	UF : 0, UT : 6,		CONFIG : 'N U T, 0, 0, 0',
	X =  474.797  mm,	Y =   -334.589  mm,	Z =   -248.128  mm,
	W =  90.000 deg,	P =   0.000 deg,	R =   90.000 deg
};
P[1529]{
   GP1:
	UF : 0, UT : 6,		CONFIG : 'N U T, 0, 0, 0',
	X =  474.358  mm,	Y =   -333.597  mm,	Z =   -247.804  mm,
	W =  90.000 deg,	P =   0.000 deg,	R =   90.000 deg
};
P[1530]{
   GP1:
	UF : 0, UT : 6,		CONFIG : 'N U T, 0, 0, 0',
	X =  473.486  mm,	Y =   -332.265  mm,	Z =   -248.052  mm,
	W =  90.000 deg,	P =   0.000 deg,	R =   90.000 deg
};
P[1531]{
   GP1:
	UF : 0, UT : 6,		CONFIG : 'N U T, 0, 0, 0',
	X =  472.911  mm,	Y =   -331.359  mm,	Z =   -248.179  mm,
	W =  90.000 deg,	P =   0.000 deg,	R =   90.000 deg
};
P[1532]{
   GP1:
	UF : 0, UT : 6,		CONFIG : 'N U T, 0, 0, 0',
	X =  472.436  mm,	Y =   -330.414  mm,	Z =   -248.006  mm,
	W =  90.000 deg,	P =   0.000 deg,	R =   90.000 deg
};
P[1533]{
   GP1:
	UF : 0, UT : 6,		CONFIG : 'N U T, 0, 0, 0',
	X =  470.822  mm,	Y =   -327.714  mm,	Z =   -248.142  mm,
	W =  90.000 deg,	P =   0.000 deg,	R =   90.000 deg
};
P[1534]{
   GP1:
	UF : 0, UT : 6,		CONFIG : 'N U T, 0, 0, 0',
	X =  470.360  mm,	Y =   -326.792  mm,	Z =   -247.970  mm,
	W =  90.000 deg,	P =   0.000 deg,	R =   90.000 deg
};
P[1535]{
   GP1:
	UF : 0, UT : 6,		CONFIG : 'N U T, 0, 0, 0',
	X =  469.532  mm,	Y =   -325.400  mm,	Z =   -248.029  mm,
	W =  90.000 deg,	P =   0.000 deg,	R =   90.000 deg
};
P[1536]{
   GP1:
	UF : 0, UT : 6,		CONFIG : 'N U T, 0, 0, 0',
	X =  468.396  mm,	Y =   -323.373  mm,	Z =   -247.945  mm,
	W =  90.000 deg,	P =   0.000 deg,	R =   90.000 deg
};
P[1537]{
   GP1:
	UF : 0, UT : 6,		CONFIG : 'N U T, 0, 0, 0',
	X =  467.953  mm,	Y =   -322.646  mm,	Z =   -248.001  mm,
	W =  90.000 deg,	P =   0.000 deg,	R =   90.000 deg
};
P[1538]{
   GP1:
	UF : 0, UT : 6,		CONFIG : 'N U T, 0, 0, 0',
	X =  467.093  mm,	Y =   -321.165  mm,	Z =   -248.010  mm,
	W =  90.000 deg,	P =   0.000 deg,	R =   90.000 deg
};
P[1539]{
   GP1:
	UF : 0, UT : 6,		CONFIG : 'N U T, 0, 0, 0',
	X =  465.613  mm,	Y =   -318.699  mm,	Z =   -248.148  mm,
	W =  90.000 deg,	P =   0.000 deg,	R =   90.000 deg
};
P[1540]{
   GP1:
	UF : 0, UT : 6,		CONFIG : 'N U T, 0, 0, 0',
	X =  464.567  mm,	Y =   -316.920  mm,	Z =   -248.196  mm,
	W =  90.000 deg,	P =   0.000 deg,	R =   90.000 deg
};
P[1541]{
   GP1:
	UF : 0, UT : 6,		CONFIG : 'N U T, 0, 0, 0',
	X =  463.631  mm,	Y =   -315.161  mm,	Z =   -248.002  mm,
	W =  90.000 deg,	P =   0.000 deg,	R =   90.000 deg
};
P[1542]{
   GP1:
	UF : 0, UT : 6,		CONFIG : 'N U T, 0, 0, 0',
	X =  463.100  mm,	Y =   -314.216  mm,	Z =   -247.965  mm,
	W =  90.000 deg,	P =   0.000 deg,	R =   90.000 deg
};
P[1543]{
   GP1:
	UF : 0, UT : 6,		CONFIG : 'N U T, 0, 0, 0',
	X =  462.160  mm,	Y =   -312.535  mm,	Z =   -247.892  mm,
	W =  90.000 deg,	P =   0.000 deg,	R =   90.000 deg
};
P[1544]{
   GP1:
	UF : 0, UT : 6,		CONFIG : 'N U T, 0, 0, 0',
	X =  461.282  mm,	Y =   -311.005  mm,	Z =   -247.880  mm,
	W =  90.000 deg,	P =   0.000 deg,	R =   90.000 deg
};
P[1545]{
   GP1:
	UF : 0, UT : 6,		CONFIG : 'N U T, 0, 0, 0',
	X =  460.643  mm,	Y =   -310.130  mm,	Z =   -248.205  mm,
	W =  90.000 deg,	P =   0.000 deg,	R =   90.000 deg
};
P[1546]{
   GP1:
	UF : 0, UT : 6,		CONFIG : 'N U T, 0, 0, 0',
	X =  458.837  mm,	Y =   -307.025  mm,	Z =   -248.237  mm,
	W =  90.000 deg,	P =   0.000 deg,	R =   90.000 deg
};
P[1547]{
   GP1:
	UF : 0, UT : 6,		CONFIG : 'N U T, 0, 0, 0',
	X =  457.547  mm,	Y =   -304.731  mm,	Z =   -248.150  mm,
	W =  90.000 deg,	P =   0.000 deg,	R =   90.000 deg
};
P[1548]{
   GP1:
	UF : 0, UT : 6,		CONFIG : 'N U T, 0, 0, 0',
	X =  456.867  mm,	Y =   -303.518  mm,	Z =   -248.103  mm,
	W =  90.000 deg,	P =   0.000 deg,	R =   90.000 deg
};
P[1549]{
   GP1:
	UF : 0, UT : 6,		CONFIG : 'N U T, 0, 0, 0',
	X =  455.788  mm,	Y =   -301.711  mm,	Z =   -248.187  mm,
	W =  90.000 deg,	P =   0.000 deg,	R =   90.000 deg
};
P[1550]{
   GP1:
	UF : 0, UT : 6,		CONFIG : 'N U T, 0, 0, 0',
	X =  454.454  mm,	Y =   -299.407  mm,	Z =   -248.197  mm,
	W =  90.000 deg,	P =   0.000 deg,	R =   90.000 deg
};
P[1551]{
   GP1:
	UF : 0, UT : 6,		CONFIG : 'N U T, 0, 0, 0',
	X =  453.882  mm,	Y =   -298.356  mm,	Z =   -248.113  mm,
	W =  90.000 deg,	P =   0.000 deg,	R =   90.000 deg
};
P[1552]{
   GP1:
	UF : 0, UT : 6,		CONFIG : 'N U T, 0, 0, 0',
	X =  453.477  mm,	Y =   -297.544  mm,	Z =   -247.960  mm,
	W =  90.000 deg,	P =   0.000 deg,	R =   90.000 deg
};
P[1553]{
   GP1:
	UF : 0, UT : 6,		CONFIG : 'N U T, 0, 0, 0',
	X =  452.176  mm,	Y =   -295.442  mm,	Z =   -248.171  mm,
	W =  90.000 deg,	P =   0.000 deg,	R =   90.000 deg
};
P[1554]{
   GP1:
	UF : 0, UT : 6,		CONFIG : 'N U T, 0, 0, 0',
	X =  451.411  mm,	Y =   -294.155  mm,	Z =   -248.222  mm,
	W =  90.000 deg,	P =   0.000 deg,	R =   90.000 deg
};
P[1555]{
   GP1:
	UF : 0, UT : 6,		CONFIG : 'N U T, 0, 0, 0',
	X =  450.241  mm,	Y =   -291.952  mm,	Z =   -247.976  mm,
	W =  90.000 deg,	P =   0.000 deg,	R =   90.000 deg
};
P[1556]{
   GP1:
	UF : 0, UT : 6,		CONFIG : 'N U T, 0, 0, 0',
	X =  449.232  mm,	Y =   -290.232  mm,	Z =   -248.015  mm,
	W =  90.000 deg,	P =   0.000 deg,	R =   90.000 deg
};
P[1557]{
   GP1:
	UF : 0, UT : 6,		CONFIG : 'N U T, 0, 0, 0',
	X =  448.784  mm,	Y =   -289.434  mm,	Z =   -247.984  mm,
	W =  90.000 deg,	P =   0.000 deg,	R =   90.000 deg
};
P[1558]{
   GP1:
	UF : 0, UT : 6,		CONFIG : 'N U T, 0, 0, 0',
	X =  447.902  mm,	Y =   -288.033  mm,	Z =   -248.160  mm,
	W =  90.000 deg,	P =   0.000 deg,	R =   90.000 deg
};
P[1559]{
   GP1:
	UF : 0, UT : 6,		CONFIG : 'N U T, 0, 0, 0',
	X =  447.571  mm,	Y =   -287.324  mm,	Z =   -247.969  mm,
	W =  90.000 deg,	P =   0.000 deg,	R =   90.000 deg
};
P[1560]{
   GP1:
	UF : 0, UT : 6,		CONFIG : 'N U T, 0, 0, 0',
	X =  445.908  mm,	Y =   -284.546  mm,	Z =   -248.113  mm,
	W =  90.000 deg,	P =   0.000 deg,	R =   90.000 deg
};
P[1561]{
   GP1:
	UF : 0, UT : 6,		CONFIG : 'N U T, 0, 0, 0',
	X =  444.581  mm,	Y =   -282.266  mm,	Z =   -248.139  mm,
	W =  90.000 deg,	P =   0.000 deg,	R =   90.000 deg
};
P[1562]{
   GP1:
	UF : 0, UT : 6,		CONFIG : 'N U T, 0, 0, 0',
	X =  443.765  mm,	Y =   -280.901  mm,	Z =   -248.206  mm,
	W =  90.000 deg,	P =   0.000 deg,	R =   90.000 deg
};
P[1563]{
   GP1:
	UF : 0, UT : 6,		CONFIG : 'N U T, 0, 0, 0',
	X =  442.689  mm,	Y =   -278.918  mm,	Z =   -248.039  mm,
	W =  90.000 deg,	P =   0.000 deg,	R =   90.000 deg
};
P[1564]{
   GP1:
	UF : 0, UT : 6,		CONFIG : 'N U T, 0, 0, 0',
	X =  441.741  mm,	Y =   -277.187  mm,	Z =   -247.917  mm,
	W =  90.000 deg,	P =   0.000 deg,	R =   90.000 deg
};
P[1565]{
   GP1:
	UF : 0, UT : 6,		CONFIG : 'N U T, 0, 0, 0',
	X =  441.319  mm,	Y =   -276.589  mm,	Z =   -248.103  mm,
	W =  90.000 deg,	P =   0.000 deg,	R =   90.000 deg
};
P[1566]{
   GP1:
	UF : 0, UT : 6,		CONFIG : 'N U T, 0, 0, 0',
	X =  440.661  mm,	Y =   -275.265  mm,	Z =   -247.842  mm,
	W =  90.000 deg,	P =   0.000 deg,	R =   90.000 deg
};
P[1567]{
   GP1:
	UF : 0, UT : 6,		CONFIG : 'N U T, 0, 0, 0',
	X =  439.825  mm,	Y =   -273.885  mm,	Z =   -247.936  mm,
	W =  90.000 deg,	P =   0.000 deg,	R =   90.000 deg
};
P[1568]{
   GP1:
	UF : 0, UT : 6,		CONFIG : 'N U T, 0, 0, 0',
	X =  437.965  mm,	Y =   -270.714  mm,	Z =   -248.009  mm,
	W =  90.000 deg,	P =   0.000 deg,	R =   90.000 deg
};
P[1569]{
   GP1:
	UF : 0, UT : 6,		CONFIG : 'N U T, 0, 0, 0',
	X =  437.402  mm,	Y =   -269.770  mm,	Z =   -248.054  mm,
	W =  90.000 deg,	P =   0.000 deg,	R =   90.000 deg
};
P[1570]{
   GP1:
	UF : 0, UT : 6,		CONFIG : 'N U T, 0, 0, 0',
	X =  436.666  mm,	Y =   -268.332  mm,	Z =   -247.824  mm,
	W =  90.000 deg,	P =   0.000 deg,	R =   90.000 deg
};
P[1571]{
   GP1:
	UF : 0, UT : 6,		CONFIG : 'N U T, 0, 0, 0',
	X =  434.809  mm,	Y =   -265.157  mm,	Z =   -247.879  mm,
	W =  90.000 deg,	P =   0.000 deg,	R =   90.000 deg
};
P[1572]{
   GP1:
	UF : 0, UT : 6,		CONFIG : 'N U T, 0, 0, 0',
	X =  433.786  mm,	Y =   -263.608  mm,	Z =   -248.191  mm,
	W =  90.000 deg,	P =   0.000 deg,	R =   90.000 deg
};
P[1573]{
   GP1:
	UF : 0, UT : 6,		CONFIG : 'N U T, 0, 0, 0',
	X =  431.779  mm,	Y =   -260.065  mm,	Z =   -248.099  mm,
	W =  90.000 deg,	P =   0.000 deg,	R =   90.000 deg
};
P[1574]{
   GP1:
	UF : 0, UT : 6,		CONFIG : 'N U T, 0, 0, 0',
	X =  430.861  mm,	Y =   -258.520  mm,	Z =   -248.160  mm,
	W =  90.000 deg,	P =   0.000 deg,	R =   90.000 deg
};
P[1575]{
   GP1:
	UF : 0, UT : 6,		CONFIG : 'N U T, 0, 0, 0',
	X =  429.870  mm,	Y =   -256.679  mm,	Z =   -247.988  mm,
	W =  90.000 deg,	P =   0.000 deg,	R =   90.000 deg
};
P[1576]{
   GP1:
	UF : 0, UT : 6,		CONFIG : 'N U T, 0, 0, 0',
	X =  429.103  mm,	Y =   -255.377  mm,	Z =   -248.023  mm,
	W =  90.000 deg,	P =   0.000 deg,	R =   90.000 deg
};
P[1577]{
   GP1:
	UF : 0, UT : 6,		CONFIG : 'N U T, 0, 0, 0',
	X =  427.799  mm,	Y =   -253.282  mm,	Z =   -248.252  mm,
	W =  90.000 deg,	P =   0.000 deg,	R =   90.000 deg
};
P[1578]{
   GP1:
	UF : 0, UT : 6,		CONFIG : 'N U T, 0, 0, 0',
	X =  426.471  mm,	Y =   -250.902  mm,	Z =   -248.142  mm,
	W =  90.000 deg,	P =   0.000 deg,	R =   90.000 deg
};
P[1579]{
   GP1:
	UF : 0, UT : 6,		CONFIG : 'N U T, 0, 0, 0',
	X =  424.128  mm,	Y =   -246.770  mm,	Z =   -248.038  mm,
	W =  90.000 deg,	P =   0.000 deg,	R =   90.000 deg
};
P[1580]{
   GP1:
	UF : 0, UT : 6,		CONFIG : 'N U T, 0, 0, 0',
	X =  423.540  mm,	Y =   -245.657  mm,	Z =   -247.904  mm,
	W =  90.000 deg,	P =   0.000 deg,	R =   90.000 deg
};
P[1581]{
   GP1:
	UF : 0, UT : 6,		CONFIG : 'N U T, 0, 0, 0',
	X =  422.892  mm,	Y =   -244.754  mm,	Z =   -248.213  mm,
	W =  90.000 deg,	P =   0.000 deg,	R =   90.000 deg
};
P[1582]{
   GP1:
	UF : 0, UT : 6,		CONFIG : 'N U T, 0, 0, 0',
	X =  422.474  mm,	Y =   -243.890  mm,	Z =   -248.015  mm,
	W =  90.000 deg,	P =   0.000 deg,	R =   90.000 deg
};
P[1583]{
   GP1:
	UF : 0, UT : 6,		CONFIG : 'N U T, 0, 0, 0',
	X =  421.948  mm,	Y =   -242.939  mm,	Z =   -247.959  mm,
	W =  90.000 deg,	P =   0.000 deg,	R =   90.000 deg
};
P[1584]{
   GP1:
	UF : 0, UT : 6,		CONFIG : 'N U T, 0, 0, 0',
	X =  420.779  mm,	Y =   -240.907  mm,	Z =   -247.948  mm,
	W =  90.000 deg,	P =   0.000 deg,	R =   90.000 deg
};
P[1585]{
   GP1:
	UF : 0, UT : 6,		CONFIG : 'N U T, 0, 0, 0',
	X =  419.758  mm,	Y =   -239.064  mm,	Z =   -247.845  mm,
	W =  90.000 deg,	P =   0.000 deg,	R =   90.000 deg
};
P[1586]{
   GP1:
	UF : 0, UT : 6,		CONFIG : 'N U T, 0, 0, 0',
	X =  418.658  mm,	Y =   -237.324  mm,	Z =   -248.077  mm,
	W =  90.000 deg,	P =   0.000 deg,	R =   90.000 deg
};
P[1587]{
   GP1:
	UF : 0, UT : 6,		CONFIG : 'N U T, 0, 0, 0',
	X =  417.346  mm,	Y =   -234.899  mm,	Z =   -247.861  mm,
	W =  90.000 deg,	P =   0.000 deg,	R =   90.000 deg
};
P[1588]{
   GP1:
	UF : 0, UT : 6,		CONFIG : 'N U T, 0, 0, 0',
	X =  416.514  mm,	Y =   -233.665  mm,	Z =   -248.152  mm,
	W =  90.000 deg,	P =   0.000 deg,	R =   90.000 deg
};
P[1589]{
   GP1:
	UF : 0, UT : 6,		CONFIG : 'N U T, 0, 0, 0',
	X =  414.834  mm,	Y =   -230.647  mm,	Z =   -248.001  mm,
	W =  90.000 deg,	P =   0.000 deg,	R =   90.000 deg
};
P[1590]{
   GP1:
	UF : 0, UT : 6,		CONFIG : 'N U T, 0, 0, 0',
	X =  411.599  mm,	Y =   -225.074  mm,	Z =   -248.043  mm,
	W =  90.000 deg,	P =   0.000 deg,	R =   90.000 deg
};
P[1591]{
   GP1:
	UF : 0, UT : 6,		CONFIG : 'N U T, 0, 0, 0',
	X =  410.932  mm,	Y =   -223.910  mm,	Z =   -248.028  mm,
	W =  90.000 deg,	P =   0.000 deg,	R =   90.000 deg
};
P[1592]{
   GP1:
	UF : 0, UT : 6,		CONFIG : 'N U T, 0, 0, 0',
	X =  410.483  mm,	Y =   -222.966  mm,	Z =   -247.797  mm,
	W =  90.000 deg,	P =   0.000 deg,	R =   90.000 deg
};
P[1593]{
   GP1:
	UF : 0, UT : 6,		CONFIG : 'N U T, 0, 0, 0',
	X =  410.046  mm,	Y =   -222.431  mm,	Z =   -248.109  mm,
	W =  90.000 deg,	P =   0.000 deg,	R =   90.000 deg
};
P[1594]{
   GP1:
	UF : 0, UT : 6,		CONFIG : 'N U T, 0, 0, 0',
	X =  409.035  mm,	Y =   -220.506  mm,	Z =   -247.865  mm,
	W =  90.000 deg,	P =   0.000 deg,	R =   90.000 deg
};
P[1595]{
   GP1:
	UF : 0, UT : 6,		CONFIG : 'N U T, 0, 0, 0',
	X =  408.248  mm,	Y =   -219.271  mm,	Z =   -248.042  mm,
	W =  90.000 deg,	P =   0.000 deg,	R =   90.000 deg
};
P[1596]{
   GP1:
	UF : 0, UT : 6,		CONFIG : 'N U T, 0, 0, 0',
	X =  407.871  mm,	Y =   -218.702  mm,	Z =   -248.158  mm,
	W =  90.000 deg,	P =   0.000 deg,	R =   90.000 deg
};
P[1597]{
   GP1:
	UF : 0, UT : 6,		CONFIG : 'N U T, 0, 0, 0',
	X =  407.029  mm,	Y =   -217.194  mm,	Z =   -248.092  mm,
	W =  90.000 deg,	P =   0.000 deg,	R =   90.000 deg
};
P[1598]{
   GP1:
	UF : 0, UT : 6,		CONFIG : 'N U T, 0, 0, 0',
	X =  406.712  mm,	Y =   -216.429  mm,	Z =   -247.788  mm,
	W =  90.000 deg,	P =   0.000 deg,	R =   90.000 deg
};
P[1599]{
   GP1:
	UF : 0, UT : 6,		CONFIG : 'N U T, 0, 0, 0',
	X =  405.760  mm,	Y =   -214.893  mm,	Z =   -247.947  mm,
	W =  90.000 deg,	P =   0.000 deg,	R =   90.000 deg
};
P[1600]{
   GP1:
	UF : 0, UT : 6,		CONFIG : 'N U T, 0, 0, 0',
	X =  403.495  mm,	Y =   -211.142  mm,	Z =   -248.188  mm,
	W =  90.000 deg,	P =   0.000 deg,	R =   90.000 deg
};
P[1601]{
   GP1:
	UF : 0, UT : 6,		CONFIG : 'N U T, 0, 0, 0',
	X =  401.729  mm,	Y =   -208.099  mm,	Z =   -248.209  mm,
	W =  90.000 deg,	P =   0.000 deg,	R =   90.000 deg
};
P[1602]{
   GP1:
	UF : 0, UT : 6,		CONFIG : 'N U T, 0, 0, 0',
	X =  401.215  mm,	Y =   -207.155  mm,	Z =   -248.132  mm,
	W =  90.000 deg,	P =   0.000 deg,	R =   90.000 deg
};
P[1603]{
   GP1:
	UF : 0, UT : 6,		CONFIG : 'N U T, 0, 0, 0',
	X =  400.460  mm,	Y =   -205.608  mm,	Z =   -247.798  mm,
	W =  90.000 deg,	P =   0.000 deg,	R =   90.000 deg
};
P[1604]{
   GP1:
	UF : 0, UT : 6,		CONFIG : 'N U T, 0, 0, 0',
	X =  399.951  mm,	Y =   -205.002  mm,	Z =   -248.184  mm,
	W =  90.000 deg,	P =   0.000 deg,	R =   90.000 deg
};
P[1605]{
   GP1:
	UF : 0, UT : 6,		CONFIG : 'N U T, 0, 0, 0',
	X =  398.920  mm,	Y =   -203.065  mm,	Z =   -247.973  mm,
	W =  90.000 deg,	P =   0.000 deg,	R =   90.000 deg
};
P[1606]{
   GP1:
	UF : 0, UT : 6,		CONFIG : 'N U T, 0, 0, 0',
	X =  397.944  mm,	Y =   -201.529  mm,	Z =   -248.191  mm,
	W =  90.000 deg,	P =   0.000 deg,	R =   90.000 deg
};
P[1607]{
   GP1:
	UF : 0, UT : 6,		CONFIG : 'N U T, 0, 0, 0',
	X =  396.430  mm,	Y =   -198.848  mm,	Z =   -248.106  mm,
	W =  90.000 deg,	P =   0.000 deg,	R =   90.000 deg
};
P[1608]{
   GP1:
	UF : 0, UT : 6,		CONFIG : 'N U T, 0, 0, 0',
	X =  396.083  mm,	Y =   -198.130  mm,	Z =   -247.940  mm,
	W =  90.000 deg,	P =   0.000 deg,	R =   90.000 deg
};
P[1609]{
   GP1:
	UF : 0, UT : 6,		CONFIG : 'N U T, 0, 0, 0',
	X =  395.279  mm,	Y =   -196.767  mm,	Z =   -247.982  mm,
	W =  90.000 deg,	P =   0.000 deg,	R =   90.000 deg
};
P[1610]{
   GP1:
	UF : 0, UT : 6,		CONFIG : 'N U T, 0, 0, 0',
	X =  394.631  mm,	Y =   -195.731  mm,	Z =   -248.102  mm,
	W =  90.000 deg,	P =   0.000 deg,	R =   90.000 deg
};
P[1611]{
   GP1:
	UF : 0, UT : 6,		CONFIG : 'N U T, 0, 0, 0',
	X =  392.922  mm,	Y =   -192.760  mm,	Z =   -248.088  mm,
	W =  90.000 deg,	P =   0.000 deg,	R =   90.000 deg
};
P[1612]{
   GP1:
	UF : 0, UT : 6,		CONFIG : 'N U T, 0, 0, 0',
	X =  391.251  mm,	Y =   -189.891  mm,	Z =   -248.124  mm,
	W =  90.000 deg,	P =   0.000 deg,	R =   90.000 deg
};
P[1613]{
   GP1:
	UF : 0, UT : 6,		CONFIG : 'N U T, 0, 0, 0',
	X =  388.461  mm,	Y =   -184.918  mm,	Z =   -247.925  mm,
	W =  90.000 deg,	P =   0.000 deg,	R =   90.000 deg
};
P[1614]{
   GP1:
	UF : 0, UT : 6,		CONFIG : 'N U T, 0, 0, 0',
	X =  387.068  mm,	Y =   -182.568  mm,	Z =   -248.014  mm,
	W =  90.000 deg,	P =   0.000 deg,	R =   90.000 deg
};
P[1615]{
   GP1:
	UF : 0, UT : 6,		CONFIG : 'N U T, 0, 0, 0',
	X =  386.082  mm,	Y =   -180.926  mm,	Z =   -248.105  mm,
	W =  90.000 deg,	P =   0.000 deg,	R =   90.000 deg
};
P[1616]{
   GP1:
	UF : 0, UT : 6,		CONFIG : 'N U T, 0, 0, 0',
	X =  385.512  mm,	Y =   -179.717  mm,	Z =   -247.796  mm,
	W =  90.000 deg,	P =   0.000 deg,	R =   90.000 deg
};
P[1617]{
   GP1:
	UF : 0, UT : 6,		CONFIG : 'N U T, 0, 0, 0',
	X =  385.093  mm,	Y =   -179.000  mm,	Z =   -247.806  mm,
	W =  90.000 deg,	P =   0.000 deg,	R =   90.000 deg
};
P[1618]{
   GP1:
	UF : 0, UT : 6,		CONFIG : 'N U T, 0, 0, 0',
	X =  383.900  mm,	Y =   -177.145  mm,	Z =   -248.103  mm,
	W =  90.000 deg,	P =   0.000 deg,	R =   90.000 deg
};
P[1619]{
   GP1:
	UF : 0, UT : 6,		CONFIG : 'N U T, 0, 0, 0',
	X =  382.403  mm,	Y =   -174.331  mm,	Z =   -247.792  mm,
	W =  90.000 deg,	P =   0.000 deg,	R =   90.000 deg
};
P[1620]{
   GP1:
	UF : 0, UT : 6,		CONFIG : 'N U T, 0, 0, 0',
	X =  381.568  mm,	Y =   -173.118  mm,	Z =   -248.120  mm,
	W =  90.000 deg,	P =   0.000 deg,	R =   90.000 deg
};
P[1621]{
   GP1:
	UF : 0, UT : 6,		CONFIG : 'N U T, 0, 0, 0',
	X =  381.064  mm,	Y =   -172.155  mm,	Z =   -247.994  mm,
	W =  90.000 deg,	P =   0.000 deg,	R =   90.000 deg
};
P[1622]{
   GP1:
	UF : 0, UT : 6,		CONFIG : 'N U T, 0, 0, 0',
	X =  380.600  mm,	Y =   -171.355  mm,	Z =   -247.998  mm,
	W =  90.000 deg,	P =   0.000 deg,	R =   90.000 deg
};
P[1623]{
   GP1:
	UF : 0, UT : 6,		CONFIG : 'N U T, 0, 0, 0',
	X =  378.626  mm,	Y =   -168.094  mm,	Z =   -248.218  mm,
	W =  90.000 deg,	P =   0.000 deg,	R =   90.000 deg
};
P[1624]{
   GP1:
	UF : 0, UT : 6,		CONFIG : 'N U T, 0, 0, 0',
	X =  377.762  mm,	Y =   -166.420  mm,	Z =   -247.969  mm,
	W =  90.000 deg,	P =   0.000 deg,	R =   90.000 deg
};
P[1625]{
   GP1:
	UF : 0, UT : 6,		CONFIG : 'N U T, 0, 0, 0',
	X =  376.901  mm,	Y =   -164.970  mm,	Z =   -248.028  mm,
	W =  90.000 deg,	P =   0.000 deg,	R =   90.000 deg
};
P[1626]{
   GP1:
	UF : 0, UT : 6,		CONFIG : 'N U T, 0, 0, 0',
	X =  376.473  mm,	Y =   -164.173  mm,	Z =   -247.952  mm,
	W =  90.000 deg,	P =   0.000 deg,	R =   90.000 deg
};
P[1627]{
   GP1:
	UF : 0, UT : 6,		CONFIG : 'N U T, 0, 0, 0',
	X =  375.645  mm,	Y =   -162.611  mm,	Z =   -247.770  mm,
	W =  90.000 deg,	P =   0.000 deg,	R =   90.000 deg
};
P[1628]{
   GP1:
	UF : 0, UT : 6,		CONFIG : 'N U T, 0, 0, 0',
	X =  375.141  mm,	Y =   -162.012  mm,	Z =   -248.154  mm,
	W =  90.000 deg,	P =   0.000 deg,	R =   90.000 deg
};
P[1629]{
   GP1:
	UF : 0, UT : 6,		CONFIG : 'N U T, 0, 0, 0',
	X =  374.441  mm,	Y =   -160.590  mm,	Z =   -247.861  mm,
	W =  90.000 deg,	P =   0.000 deg,	R =   90.000 deg
};
P[1630]{
   GP1:
	UF : 0, UT : 6,		CONFIG : 'N U T, 0, 0, 0',
	X =  372.124  mm,	Y =   -156.753  mm,	Z =   -248.107  mm,
	W =  90.000 deg,	P =   0.000 deg,	R =   90.000 deg
};
P[1631]{
   GP1:
	UF : 0, UT : 6,		CONFIG : 'N U T, 0, 0, 0',
	X =  371.314  mm,	Y =   -155.317  mm,	Z =   -248.062  mm,
	W =  90.000 deg,	P =   0.000 deg,	R =   90.000 deg
};
P[1632]{
   GP1:
	UF : 0, UT : 6,		CONFIG : 'N U T, 0, 0, 0',
	X =  370.225  mm,	Y =   -153.429  mm,	Z =   -248.057  mm,
	W =  90.000 deg,	P =   0.000 deg,	R =   90.000 deg
};
P[1633]{
   GP1:
	UF : 0, UT : 6,		CONFIG : 'N U T, 0, 0, 0',
	X =  369.441  mm,	Y =   -151.898  mm,	Z =   -247.814  mm,
	W =  90.000 deg,	P =   0.000 deg,	R =   90.000 deg
};
P[1634]{
   GP1:
	UF : 0, UT : 6,		CONFIG : 'N U T, 0, 0, 0',
	X =  367.319  mm,	Y =   -148.417  mm,	Z =   -248.088  mm,
	W =  90.000 deg,	P =   0.000 deg,	R =   90.000 deg
};
P[1635]{
   GP1:
	UF : 0, UT : 6,		CONFIG : 'N U T, 0, 0, 0',
	X =  366.654  mm,	Y =   -147.274  mm,	Z =   -248.100  mm,
	W =  90.000 deg,	P =   0.000 deg,	R =   90.000 deg
};
P[1636]{
   GP1:
	UF : 0, UT : 6,		CONFIG : 'N U T, 0, 0, 0',
	X =  365.710  mm,	Y =   -145.408  mm,	Z =   -247.778  mm,
	W =  90.000 deg,	P =   0.000 deg,	R =   90.000 deg
};
P[1637]{
   GP1:
	UF : 0, UT : 6,		CONFIG : 'N U T, 0, 0, 0',
	X =  364.963  mm,	Y =   -144.240  mm,	Z =   -247.951  mm,
	W =  90.000 deg,	P =   0.000 deg,	R =   90.000 deg
};
P[1638]{
   GP1:
	UF : 0, UT : 6,		CONFIG : 'N U T, 0, 0, 0',
	X =  362.252  mm,	Y =   -139.569  mm,	Z =   -247.988  mm,
	W =  90.000 deg,	P =   0.000 deg,	R =   90.000 deg
};
P[1639]{
   GP1:
	UF : 0, UT : 6,		CONFIG : 'N U T, 0, 0, 0',
	X =  360.992  mm,	Y =   -137.293  mm,	Z =   -247.856  mm,
	W =  90.000 deg,	P =   0.000 deg,	R =   90.000 deg
};
P[1640]{
   GP1:
	UF : 0, UT : 6,		CONFIG : 'N U T, 0, 0, 0',
	X =  359.863  mm,	Y =   -135.498  mm,	Z =   -248.080  mm,
	W =  90.000 deg,	P =   0.000 deg,	R =   90.000 deg
};
P[1641]{
   GP1:
	UF : 0, UT : 6,		CONFIG : 'N U T, 0, 0, 0',
	X =  359.474  mm,	Y =   -134.912  mm,	Z =   -248.205  mm,
	W =  90.000 deg,	P =   0.000 deg,	R =   90.000 deg
};
P[1642]{
   GP1:
	UF : 0, UT : 6,		CONFIG : 'N U T, 0, 0, 0',
	X =  358.888  mm,	Y =   -133.873  mm,	Z =   -248.168  mm,
	W =  90.000 deg,	P =   0.000 deg,	R =   90.000 deg
};
P[1643]{
   GP1:
	UF : 0, UT : 6,		CONFIG : 'N U T, 0, 0, 0',
	X =  358.663  mm,	Y =   -133.250  mm,	Z =   -247.841  mm,
	W =  90.000 deg,	P =   0.000 deg,	R =   90.000 deg
};
P[1644]{
   GP1:
	UF : 0, UT : 6,		CONFIG : 'N U T, 0, 0, 0',
	X =  357.355  mm,	Y =   -131.276  mm,	Z =   -248.250  mm,
	W =  90.000 deg,	P =   0.000 deg,	R =   90.000 deg
};
P[1645]{
   GP1:
	UF : 0, UT : 6,		CONFIG : 'N U T, 0, 0, 0',
	X =  357.087  mm,	Y =   -130.536  mm,	Z =   -247.863  mm,
	W =  90.000 deg,	P =   0.000 deg,	R =   90.000 deg
};
P[1646]{
   GP1:
	UF : 0, UT : 6,		CONFIG : 'N U T, 0, 0, 0',
	X =  355.787  mm,	Y =   -128.521  mm,	Z =   -248.196  mm,
	W =  90.000 deg,	P =   0.000 deg,	R =   90.000 deg
};
P[1647]{
   GP1:
	UF : 0, UT : 6,		CONFIG : 'N U T, 0, 0, 0',
	X =  355.163  mm,	Y =   -127.365  mm,	Z =   -248.088  mm,
	W =  90.000 deg,	P =   0.000 deg,	R =   90.000 deg
};
P[1648]{
   GP1:
	UF : 0, UT : 6,		CONFIG : 'N U T, 0, 0, 0',
	X =  354.057  mm,	Y =   -125.533  mm,	Z =   -248.207  mm,
	W =  90.000 deg,	P =   0.000 deg,	R =   90.000 deg
};
P[1649]{
   GP1:
	UF : 0, UT : 6,		CONFIG : 'N U T, 0, 0, 0',
	X =  352.390  mm,	Y =   -122.837  mm,	Z =   -248.021  mm,
	W =  90.000 deg,	P =   0.000 deg,	R =   90.000 deg
};
P[1650]{
   GP1:
	UF : 0, UT : 6,		CONFIG : 'N U T, 0, 0, 0',
	X =  351.347  mm,	Y =   -121.500  mm,	Z =   -248.021  mm,
	W =  90.000 deg,	P =   0.000 deg,	R =   90.000 deg
};
P[1651]{
   GP1:
	UF : 0, UT : 6,		CONFIG : 'N U T, 0, 0, 0',
	X =  350.186  mm,	Y =   -120.520  mm,	Z =   -248.165  mm,
	W =  90.000 deg,	P =   0.000 deg,	R =   90.000 deg
};
P[1652]{
   GP1:
	UF : 0, UT : 6,		CONFIG : 'N U T, 0, 0, 0',
	X =  348.058  mm,	Y =   -119.038  mm,	Z =   -248.228  mm,
	W =  90.000 deg,	P =   0.000 deg,	R =   90.000 deg
};
P[1653]{
   GP1:
	UF : 0, UT : 6,		CONFIG : 'N U T, 0, 0, 0',
	X =  347.412  mm,	Y =   -118.671  mm,	Z =   -248.193  mm,
	W =  90.000 deg,	P =   0.000 deg,	R =   90.000 deg
};
P[1654]{
   GP1:
	UF : 0, UT : 6,		CONFIG : 'N U T, 0, 0, 0',
	X =  346.565  mm,	Y =   -118.157  mm,	Z =   -248.036  mm,
	W =  90.000 deg,	P =   0.000 deg,	R =   90.000 deg
};
P[1655]{
   GP1:
	UF : 0, UT : 6,		CONFIG : 'N U T, 0, 0, 0',
	X =  342.539  mm,	Y =   -117.314  mm,	Z =   -248.191  mm,
	W =  90.000 deg,	P =   0.000 deg,	R =   90.000 deg
};
P[1656]{
   GP1:
	UF : 0, UT : 6,		CONFIG : 'N U T, 0, 0, 0',
	X =  341.612  mm,	Y =   -117.227  mm,	Z =   -248.068  mm,
	W =  90.000 deg,	P =   0.000 deg,	R =   90.000 deg
};
P[1657]{
   GP1:
	UF : 0, UT : 6,		CONFIG : 'N U T, 0, 0, 0',
	X =  340.608  mm,	Y =   -117.192  mm,	Z =   -247.999  mm,
	W =  90.000 deg,	P =   0.000 deg,	R =   90.000 deg
};
P[1658]{
   GP1:
	UF : 0, UT : 6,		CONFIG : 'N U T, 0, 0, 0',
	X =  339.673  mm,	Y =   -117.287  mm,	Z =   -247.946  mm,
	W =  90.000 deg,	P =   0.000 deg,	R =   90.000 deg
};
P[1659]{
   GP1:
	UF : 0, UT : 6,		CONFIG : 'N U T, 0, 0, 0',
	X =  338.716  mm,	Y =   -117.545  mm,	Z =   -248.088  mm,
	W =  90.000 deg,	P =   0.000 deg,	R =   90.000 deg
};
P[1660]{
   GP1:
	UF : 0, UT : 6,		CONFIG : 'N U T, 0, 0, 0',
	X =  335.442  mm,	Y =   -118.670  mm,	Z =   -248.077  mm,
	W =  90.000 deg,	P =   0.000 deg,	R =   90.000 deg
};
P[1661]{
   GP1:
	UF : 0, UT : 6,		CONFIG : 'N U T, 0, 0, 0',
	X =  332.275  mm,	Y =   -120.379  mm,	Z =   -248.080  mm,
	W =  90.000 deg,	P =   0.000 deg,	R =   90.000 deg
};
P[1662]{
   GP1:
	UF : 0, UT : 6,		CONFIG : 'N U T, 0, 0, 0',
	X =  330.761  mm,	Y =   -121.280  mm,	Z =   -248.144  mm,
	W =  90.000 deg,	P =   0.000 deg,	R =   90.000 deg
};
P[1663]{
   GP1:
	UF : 0, UT : 6,		CONFIG : 'N U T, 0, 0, 0',
	X =  329.485  mm,	Y =   -121.973  mm,	Z =   -248.039  mm,
	W =  90.000 deg,	P =   0.000 deg,	R =   90.000 deg
};
P[1664]{
   GP1:
	UF : 0, UT : 6,		CONFIG : 'N U T, 0, 0, 0',
	X =  328.554  mm,	Y =   -122.548  mm,	Z =   -248.129  mm,
	W =  90.000 deg,	P =   0.000 deg,	R =   90.000 deg
};
P[1665]{
   GP1:
	UF : 0, UT : 6,		CONFIG : 'N U T, 0, 0, 0',
	X =  327.835  mm,	Y =   -122.827  mm,	Z =   -247.797  mm,
	W =  90.000 deg,	P =   0.000 deg,	R =   90.000 deg
};
P[1666]{
   GP1:
	UF : 0, UT : 6,		CONFIG : 'N U T, 0, 0, 0',
	X =  326.759  mm,	Y =   -123.439  mm,	Z =   -247.778  mm,
	W =  90.000 deg,	P =   0.000 deg,	R =   90.000 deg
};
P[1667]{
   GP1:
	UF : 0, UT : 6,		CONFIG : 'N U T, 0, 0, 0',
	X =  325.015  mm,	Y =   -124.510  mm,	Z =   -247.931  mm,
	W =  90.000 deg,	P =   0.000 deg,	R =   90.000 deg
};
P[1668]{
   GP1:
	UF : 0, UT : 6,		CONFIG : 'N U T, 0, 0, 0',
	X =  324.049  mm,	Y =   -125.182  mm,	Z =   -248.210  mm,
	W =  90.000 deg,	P =   0.000 deg,	R =   90.000 deg
};
P[1669]{
   GP1:
	UF : 0, UT : 6,		CONFIG : 'N U T, 0, 0, 0',
	X =  322.699  mm,	Y =   -125.917  mm,	Z =   -248.101  mm,
	W =  90.000 deg,	P =   0.000 deg,	R =   90.000 deg
};
P[1670]{
   GP1:
	UF : 0, UT : 6,		CONFIG : 'N U T, 0, 0, 0',
	X =  321.231  mm,	Y =   -126.639  mm,	Z =   -247.796  mm,
	W =  90.000 deg,	P =   0.000 deg,	R =   90.000 deg
};
P[1671]{
   GP1:
	UF : 0, UT : 6,		CONFIG : 'N U T, 0, 0, 0',
	X =  319.711  mm,	Y =   -127.639  mm,	Z =   -248.093  mm,
	W =  90.000 deg,	P =   0.000 deg,	R =   90.000 deg
};
P[1672]{
   GP1:
	UF : 0, UT : 6,		CONFIG : 'N U T, 0, 0, 0',
	X =  318.809  mm,	Y =   -128.158  mm,	Z =   -248.088  mm,
	W =  90.000 deg,	P =   0.000 deg,	R =   90.000 deg
};
P[1673]{
   GP1:
	UF : 0, UT : 6,		CONFIG : 'N U T, 0, 0, 0',
	X =  318.022  mm,	Y =   -128.520  mm,	Z =   -247.865  mm,
	W =  90.000 deg,	P =   0.000 deg,	R =   90.000 deg
};
P[1674]{
   GP1:
	UF : 0, UT : 6,		CONFIG : 'N U T, 0, 0, 0',
	X =  316.976  mm,	Y =   -129.207  mm,	Z =   -248.065  mm,
	W =  90.000 deg,	P =   0.000 deg,	R =   90.000 deg
};
P[1675]{
   GP1:
	UF : 0, UT : 6,		CONFIG : 'N U T, 0, 0, 0',
	X =  315.323  mm,	Y =   -130.175  mm,	Z =   -248.098  mm,
	W =  90.000 deg,	P =   0.000 deg,	R =   90.000 deg
};
P[1676]{
   GP1:
	UF : 0, UT : 6,		CONFIG : 'N U T, 0, 0, 0',
	X =  314.069  mm,	Y =   -130.782  mm,	Z =   -247.815  mm,
	W =  90.000 deg,	P =   0.000 deg,	R =   90.000 deg
};
P[1677]{
   GP1:
	UF : 0, UT : 6,		CONFIG : 'N U T, 0, 0, 0',
	X =  311.943  mm,	Y =   -132.171  mm,	Z =   -248.208  mm,
	W =  90.000 deg,	P =   0.000 deg,	R =   90.000 deg
};
P[1678]{
   GP1:
	UF : 0, UT : 6,		CONFIG : 'N U T, 0, 0, 0',
	X =  310.490  mm,	Y =   -132.831  mm,	Z =   -247.774  mm,
	W =  90.000 deg,	P =   0.000 deg,	R =   90.000 deg
};
P[1679]{
   GP1:
	UF : 0, UT : 6,		CONFIG : 'N U T, 0, 0, 0',
	X =  308.252  mm,	Y =   -134.162  mm,	Z =   -247.866  mm,
	W =  90.000 deg,	P =   0.000 deg,	R =   90.000 deg
};
P[1680]{
   GP1:
	UF : 0, UT : 6,		CONFIG : 'N U T, 0, 0, 0',
	X =  306.894  mm,	Y =   -135.065  mm,	Z =   -248.156  mm,
	W =  90.000 deg,	P =   0.000 deg,	R =   90.000 deg
};
P[1681]{
   GP1:
	UF : 0, UT : 6,		CONFIG : 'N U T, 0, 0, 0',
	X =  305.688  mm,	Y =   -135.663  mm,	Z =   -247.917  mm,
	W =  90.000 deg,	P =   0.000 deg,	R =   90.000 deg
};
P[1682]{
   GP1:
	UF : 0, UT : 6,		CONFIG : 'N U T, 0, 0, 0',
	X =  303.864  mm,	Y =   -136.718  mm,	Z =   -247.920  mm,
	W =  90.000 deg,	P =   0.000 deg,	R =   90.000 deg
};
P[1683]{
   GP1:
	UF : 0, UT : 6,		CONFIG : 'N U T, 0, 0, 0',
	X =  300.976  mm,	Y =   -138.519  mm,	Z =   -248.243  mm,
	W =  90.000 deg,	P =   0.000 deg,	R =   90.000 deg
};
P[1684]{
   GP1:
	UF : 0, UT : 6,		CONFIG : 'N U T, 0, 0, 0',
	X =  299.089  mm,	Y =   -139.563  mm,	Z =   -248.137  mm,
	W =  90.000 deg,	P =   0.000 deg,	R =   90.000 deg
};
P[1685]{
   GP1:
	UF : 0, UT : 6,		CONFIG : 'N U T, 0, 0, 0',
	X =  298.251  mm,	Y =   -140.011  mm,	Z =   -248.048  mm,
	W =  90.000 deg,	P =   0.000 deg,	R =   90.000 deg
};
P[1686]{
   GP1:
	UF : 0, UT : 6,		CONFIG : 'N U T, 0, 0, 0',
	X =  297.185  mm,	Y =   -140.686  mm,	Z =   -248.193  mm,
	W =  90.000 deg,	P =   0.000 deg,	R =   90.000 deg
};
P[1687]{
   GP1:
	UF : 0, UT : 6,		CONFIG : 'N U T, 0, 0, 0',
	X =  295.724  mm,	Y =   -141.490  mm,	Z =   -248.098  mm,
	W =  90.000 deg,	P =   0.000 deg,	R =   90.000 deg
};
P[1688]{
   GP1:
	UF : 0, UT : 6,		CONFIG : 'N U T, 0, 0, 0',
	X =  294.152  mm,	Y =   -142.266  mm,	Z =   -247.777  mm,
	W =  90.000 deg,	P =   0.000 deg,	R =   90.000 deg
};
P[1689]{
   GP1:
	UF : 0, UT : 6,		CONFIG : 'N U T, 0, 0, 0',
	X =  290.669  mm,	Y =   -144.310  mm,	Z =   -247.856  mm,
	W =  90.000 deg,	P =   0.000 deg,	R =   90.000 deg
};
P[1690]{
   GP1:
	UF : 0, UT : 6,		CONFIG : 'N U T, 0, 0, 0',
	X =  289.829  mm,	Y =   -144.910  mm,	Z =   -248.136  mm,
	W =  90.000 deg,	P =   0.000 deg,	R =   90.000 deg
};
P[1691]{
   GP1:
	UF : 0, UT : 6,		CONFIG : 'N U T, 0, 0, 0',
	X =  286.982  mm,	Y =   -146.599  mm,	Z =   -248.244  mm,
	W =  90.000 deg,	P =   0.000 deg,	R =   90.000 deg
};
P[1692]{
   GP1:
	UF : 0, UT : 6,		CONFIG : 'N U T, 0, 0, 0',
	X =  286.170  mm,	Y =   -147.024  mm,	Z =   -248.138  mm,
	W =  90.000 deg,	P =   0.000 deg,	R =   90.000 deg
};
P[1693]{
   GP1:
	UF : 0, UT : 6,		CONFIG : 'N U T, 0, 0, 0',
	X =  284.432  mm,	Y =   -147.871  mm,	Z =   -247.759  mm,
	W =  90.000 deg,	P =   0.000 deg,	R =   90.000 deg
};
P[1694]{
   GP1:
	UF : 0, UT : 6,		CONFIG : 'N U T, 0, 0, 0',
	X =  282.721  mm,	Y =   -149.012  mm,	Z =   -248.130  mm,
	W =  90.000 deg,	P =   0.000 deg,	R =   90.000 deg
};
P[1695]{
   GP1:
	UF : 0, UT : 6,		CONFIG : 'N U T, 0, 0, 0',
	X =  281.491  mm,	Y =   -149.639  mm,	Z =   -247.929  mm,
	W =  90.000 deg,	P =   0.000 deg,	R =   90.000 deg
};
P[1696]{
   GP1:
	UF : 0, UT : 6,		CONFIG : 'N U T, 0, 0, 0',
	X =  278.957  mm,	Y =   -151.235  mm,	Z =   -248.252  mm,
	W =  90.000 deg,	P =   0.000 deg,	R =   90.000 deg
};
P[1697]{
   GP1:
	UF : 0, UT : 6,		CONFIG : 'N U T, 0, 0, 0',
	X =  276.387  mm,	Y =   -152.594  mm,	Z =   -247.947  mm,
	W =  90.000 deg,	P =   0.000 deg,	R =   90.000 deg
};
P[1698]{
   GP1:
	UF : 0, UT : 6,		CONFIG : 'N U T, 0, 0, 0',
	X =  275.527  mm,	Y =   -153.150  mm,	Z =   -248.093  mm,
	W =  90.000 deg,	P =   0.000 deg,	R =   90.000 deg
};
P[1699]{
   GP1:
	UF : 0, UT : 6,		CONFIG : 'N U T, 0, 0, 0',
	X =  274.546  mm,	Y =   -153.587  mm,	Z =   -247.779  mm,
	W =  90.000 deg,	P =   0.000 deg,	R =   90.000 deg
};
P[1700]{
   GP1:
	UF : 0, UT : 6,		CONFIG : 'N U T, 0, 0, 0',
	X =  273.081  mm,	Y =   -154.605  mm,	Z =   -248.195  mm,
	W =  90.000 deg,	P =   0.000 deg,	R =   90.000 deg
};
P[1701]{
   GP1:
	UF : 0, UT : 6,		CONFIG : 'N U T, 0, 0, 0',
	X =  272.043  mm,	Y =   -155.189  mm,	Z =   -248.157  mm,
	W =  90.000 deg,	P =   0.000 deg,	R =   90.000 deg
};
P[1702]{
   GP1:
	UF : 0, UT : 6,		CONFIG : 'N U T, 0, 0, 0',
	X =  270.831  mm,	Y =   -155.824  mm,	Z =   -248.002  mm,
	W =  90.000 deg,	P =   0.000 deg,	R =   90.000 deg
};
P[1703]{
   GP1:
	UF : 0, UT : 6,		CONFIG : 'N U T, 0, 0, 0',
	X =  269.506  mm,	Y =   -156.617  mm,	Z =   -248.068  mm,
	W =  90.000 deg,	P =   0.000 deg,	R =   90.000 deg
};
P[1704]{
   GP1:
	UF : 0, UT : 6,		CONFIG : 'N U T, 0, 0, 0',
	X =  268.585  mm,	Y =   -157.047  mm,	Z =   -247.825  mm,
	W =  90.000 deg,	P =   0.000 deg,	R =   90.000 deg
};
P[1705]{
   GP1:
	UF : 0, UT : 6,		CONFIG : 'N U T, 0, 0, 0',
	X =  267.197  mm,	Y =   -157.934  mm,	Z =   -248.031  mm,
	W =  90.000 deg,	P =   0.000 deg,	R =   90.000 deg
};
P[1706]{
   GP1:
	UF : 0, UT : 6,		CONFIG : 'N U T, 0, 0, 0',
	X =  265.740  mm,	Y =   -158.742  mm,	Z =   -247.948  mm,
	W =  90.000 deg,	P =   0.000 deg,	R =   90.000 deg
};
P[1707]{
   GP1:
	UF : 0, UT : 6,		CONFIG : 'N U T, 0, 0, 0',
	X =  264.975  mm,	Y =   -159.131  mm,	Z =   -247.823  mm,
	W =  90.000 deg,	P =   0.000 deg,	R =   90.000 deg
};
P[1708]{
   GP1:
	UF : 0, UT : 6,		CONFIG : 'N U T, 0, 0, 0',
	X =  264.252  mm,	Y =   -159.687  mm,	Z =   -248.158  mm,
	W =  90.000 deg,	P =   0.000 deg,	R =   90.000 deg
};
P[1709]{
   GP1:
	UF : 0, UT : 6,		CONFIG : 'N U T, 0, 0, 0',
	X =  262.334  mm,	Y =   -160.698  mm,	Z =   -247.923  mm,
	W =  90.000 deg,	P =   0.000 deg,	R =   90.000 deg
};
P[1710]{
   GP1:
	UF : 0, UT : 6,		CONFIG : 'N U T, 0, 0, 0',
	X =  258.592  mm,	Y =   -162.990  mm,	Z =   -248.243  mm,
	W =  90.000 deg,	P =   0.000 deg,	R =   90.000 deg
};
P[1711]{
   GP1:
	UF : 0, UT : 6,		CONFIG : 'N U T, 0, 0, 0',
	X =  257.211  mm,	Y =   -163.792  mm,	Z =   -248.252  mm,
	W =  90.000 deg,	P =   0.000 deg,	R =   90.000 deg
};
P[1712]{
   GP1:
	UF : 0, UT : 6,		CONFIG : 'N U T, 0, 0, 0',
	X =  255.857  mm,	Y =   -164.489  mm,	Z =   -248.048  mm,
	W =  90.000 deg,	P =   0.000 deg,	R =   90.000 deg
};
P[1713]{
   GP1:
	UF : 0, UT : 6,		CONFIG : 'N U T, 0, 0, 0',
	X =  253.967  mm,	Y =   -165.611  mm,	Z =   -248.122  mm,
	W =  90.000 deg,	P =   0.000 deg,	R =   90.000 deg
};
P[1714]{
   GP1:
	UF : 0, UT : 6,		CONFIG : 'N U T, 0, 0, 0',
	X =  252.609  mm,	Y =   -166.412  mm,	Z =   -248.165  mm,
	W =  90.000 deg,	P =   0.000 deg,	R =   90.000 deg
};
P[1715]{
   GP1:
	UF : 0, UT : 6,		CONFIG : 'N U T, 0, 0, 0',
	X =  251.120  mm,	Y =   -167.243  mm,	Z =   -248.095  mm,
	W =  90.000 deg,	P =   0.000 deg,	R =   90.000 deg
};
P[1716]{
   GP1:
	UF : 0, UT : 6,		CONFIG : 'N U T, 0, 0, 0',
	X =  244.164  mm,	Y =   -171.132  mm,	Z =   -247.783  mm,
	W =  90.000 deg,	P =   0.000 deg,	R =   90.000 deg
};
P[1717]{
   GP1:
	UF : 0, UT : 6,		CONFIG : 'N U T, 0, 0, 0',
	X =  242.968  mm,	Y =   -172.004  mm,	Z =   -248.226  mm,
	W =  90.000 deg,	P =   0.000 deg,	R =   90.000 deg
};
P[1718]{
   GP1:
	UF : 0, UT : 6,		CONFIG : 'N U T, 0, 0, 0',
	X =  241.016  mm,	Y =   -173.085  mm,	Z =   -248.113  mm,
	W =  90.000 deg,	P =   0.000 deg,	R =   90.000 deg
};
P[1719]{
   GP1:
	UF : 0, UT : 6,		CONFIG : 'N U T, 0, 0, 0',
	X =  239.118  mm,	Y =   -174.177  mm,	Z =   -248.102  mm,
	W =  90.000 deg,	P =   0.000 deg,	R =   90.000 deg
};
P[1720]{
   GP1:
	UF : 0, UT : 6,		CONFIG : 'N U T, 0, 0, 0',
	X =  238.205  mm,	Y =   -174.747  mm,	Z =   -248.209  mm,
	W =  90.000 deg,	P =   0.000 deg,	R =   90.000 deg
};
P[1721]{
   GP1:
	UF : 0, UT : 6,		CONFIG : 'N U T, 0, 0, 0',
	X =  237.371  mm,	Y =   -175.211  mm,	Z =   -248.164  mm,
	W =  90.000 deg,	P =   0.000 deg,	R =   90.000 deg
};
P[1722]{
   GP1:
	UF : 0, UT : 6,		CONFIG : 'N U T, 0, 0, 0',
	X =  236.565  mm,	Y =   -175.562  mm,	Z =   -247.889  mm,
	W =  90.000 deg,	P =   0.000 deg,	R =   90.000 deg
};
P[1723]{
   GP1:
	UF : 0, UT : 6,		CONFIG : 'N U T, 0, 0, 0',
	X =  235.671  mm,	Y =   -176.080  mm,	Z =   -247.890  mm,
	W =  90.000 deg,	P =   0.000 deg,	R =   90.000 deg
};
P[1724]{
   GP1:
	UF : 0, UT : 6,		CONFIG : 'N U T, 0, 0, 0',
	X =  234.050  mm,	Y =   -177.054  mm,	Z =   -247.986  mm,
	W =  90.000 deg,	P =   0.000 deg,	R =   90.000 deg
};
P[1725]{
   GP1:
	UF : 0, UT : 6,		CONFIG : 'N U T, 0, 0, 0',
	X =  231.004  mm,	Y =   -178.884  mm,	Z =   -248.157  mm,
	W =  90.000 deg,	P =   0.000 deg,	R =   90.000 deg
};
P[1726]{
   GP1:
	UF : 0, UT : 6,		CONFIG : 'N U T, 0, 0, 0',
	X =  229.737  mm,	Y =   -179.574  mm,	Z =   -248.057  mm,
	W =  90.000 deg,	P =   0.000 deg,	R =   90.000 deg
};
P[1727]{
   GP1:
	UF : 0, UT : 6,		CONFIG : 'N U T, 0, 0, 0',
	X =  228.016  mm,	Y =   -180.506  mm,	Z =   -247.906  mm,
	W =  90.000 deg,	P =   0.000 deg,	R =   90.000 deg
};
P[1728]{
   GP1:
	UF : 0, UT : 6,		CONFIG : 'N U T, 0, 0, 0',
	X =  222.049  mm,	Y =   -184.015  mm,	Z =   -248.062  mm,
	W =  90.000 deg,	P =   0.000 deg,	R =   90.000 deg
};
P[1729]{
   GP1:
	UF : 0, UT : 6,		CONFIG : 'N U T, 0, 0, 0',
	X =  221.158  mm,	Y =   -184.532  mm,	Z =   -248.067  mm,
	W =  90.000 deg,	P =   0.000 deg,	R =   90.000 deg
};
P[1730]{
   GP1:
	UF : 0, UT : 6,		CONFIG : 'N U T, 0, 0, 0',
	X =  220.168  mm,	Y =   -185.052  mm,	Z =   -247.939  mm,
	W =  90.000 deg,	P =   0.000 deg,	R =   90.000 deg
};
P[1731]{
   GP1:
	UF : 0, UT : 6,		CONFIG : 'N U T, 0, 0, 0',
	X =  218.710  mm,	Y =   -185.878  mm,	Z =   -247.904  mm,
	W =  90.000 deg,	P =   0.000 deg,	R =   90.000 deg
};
P[1732]{
   GP1:
	UF : 0, UT : 6,		CONFIG : 'N U T, 0, 0, 0',
	X =  216.592  mm,	Y =   -187.084  mm,	Z =   -247.860  mm,
	W =  90.000 deg,	P =   0.000 deg,	R =   90.000 deg
};
P[1733]{
   GP1:
	UF : 0, UT : 6,		CONFIG : 'N U T, 0, 0, 0',
	X =  215.880  mm,	Y =   -187.562  mm,	Z =   -248.025  mm,
	W =  90.000 deg,	P =   0.000 deg,	R =   90.000 deg
};
P[1734]{
   GP1:
	UF : 0, UT : 6,		CONFIG : 'N U T, 0, 0, 0',
	X =  213.646  mm,	Y =   -188.743  mm,	Z =   -247.760  mm,
	W =  90.000 deg,	P =   0.000 deg,	R =   90.000 deg
};
P[1735]{
   GP1:
	UF : 0, UT : 6,		CONFIG : 'N U T, 0, 0, 0',
	X =  212.326  mm,	Y =   -189.523  mm,	Z =   -247.803  mm,
	W =  90.000 deg,	P =   0.000 deg,	R =   90.000 deg
};
P[1736]{
   GP1:
	UF : 0, UT : 6,		CONFIG : 'N U T, 0, 0, 0',
	X =  211.714  mm,	Y =   -189.936  mm,	Z =   -247.949  mm,
	W =  90.000 deg,	P =   0.000 deg,	R =   90.000 deg
};
P[1737]{
   GP1:
	UF : 0, UT : 6,		CONFIG : 'N U T, 0, 0, 0',
	X =  210.606  mm,	Y =   -190.623  mm,	Z =   -248.064  mm,
	W =  90.000 deg,	P =   0.000 deg,	R =   90.000 deg
};
P[1738]{
   GP1:
	UF : 0, UT : 6,		CONFIG : 'N U T, 0, 0, 0',
	X =  209.512  mm,	Y =   -191.209  mm,	Z =   -247.954  mm,
	W =  90.000 deg,	P =   0.000 deg,	R =   90.000 deg
};
P[1739]{
   GP1:
	UF : 0, UT : 6,		CONFIG : 'N U T, 0, 0, 0',
	X =  207.701  mm,	Y =   -192.304  mm,	Z =   -248.070  mm,
	W =  90.000 deg,	P =   0.000 deg,	R =   90.000 deg
};
P[1740]{
   GP1:
	UF : 0, UT : 6,		CONFIG : 'N U T, 0, 0, 0',
	X =  206.498  mm,	Y =   -193.029  mm,	Z =   -248.146  mm,
	W =  90.000 deg,	P =   0.000 deg,	R =   90.000 deg
};
P[1741]{
   GP1:
	UF : 0, UT : 6,		CONFIG : 'N U T, 0, 0, 0',
	X =  203.854  mm,	Y =   -194.452  mm,	Z =   -247.894  mm,
	W =  90.000 deg,	P =   0.000 deg,	R =   90.000 deg
};
P[1742]{
   GP1:
	UF : 0, UT : 6,		CONFIG : 'N U T, 0, 0, 0',
	X =  202.653  mm,	Y =   -195.144  mm,	Z =   -247.891  mm,
	W =  90.000 deg,	P =   0.000 deg,	R =   90.000 deg
};
P[1743]{
   GP1:
	UF : 0, UT : 6,		CONFIG : 'N U T, 0, 0, 0',
	X =  201.022  mm,	Y =   -196.179  mm,	Z =   -248.115  mm,
	W =  90.000 deg,	P =   0.000 deg,	R =   90.000 deg
};
P[1744]{
   GP1:
	UF : 0, UT : 6,		CONFIG : 'N U T, 0, 0, 0',
	X =  200.074  mm,	Y =   -196.640  mm,	Z =   -247.908  mm,
	W =  90.000 deg,	P =   0.000 deg,	R =   90.000 deg
};
P[1745]{
   GP1:
	UF : 0, UT : 6,		CONFIG : 'N U T, 0, 0, 0',
	X =  199.042  mm,	Y =   -197.336  mm,	Z =   -248.150  mm,
	W =  90.000 deg,	P =   0.000 deg,	R =   90.000 deg
};
P[1746]{
   GP1:
	UF : 0, UT : 6,		CONFIG : 'N U T, 0, 0, 0',
	X =  198.087  mm,	Y =   -197.820  mm,	Z =   -247.988  mm,
	W =  90.000 deg,	P =   0.000 deg,	R =   90.000 deg
};
P[1747]{
   GP1:
	UF : 0, UT : 6,		CONFIG : 'N U T, 0, 0, 0',
	X =  196.694  mm,	Y =   -198.603  mm,	Z =   -247.934  mm,
	W =  90.000 deg,	P =   0.000 deg,	R =   90.000 deg
};
P[1748]{
   GP1:
	UF : 0, UT : 6,		CONFIG : 'N U T, 0, 0, 0',
	X =  194.063  mm,	Y =   -200.109  mm,	Z =   -247.906  mm,
	W =  90.000 deg,	P =   0.000 deg,	R =   90.000 deg
};
P[1749]{
   GP1:
	UF : 0, UT : 6,		CONFIG : 'N U T, 0, 0, 0',
	X =  191.490  mm,	Y =   -201.602  mm,	Z =   -247.920  mm,
	W =  90.000 deg,	P =   0.000 deg,	R =   90.000 deg
};
P[1750]{
   GP1:
	UF : 0, UT : 6,		CONFIG : 'N U T, 0, 0, 0',
	X =  190.654  mm,	Y =   -202.081  mm,	Z =   -247.913  mm,
	W =  90.000 deg,	P =   0.000 deg,	R =   90.000 deg
};
P[1751]{
   GP1:
	UF : 0, UT : 6,		CONFIG : 'N U T, 0, 0, 0',
	X =  189.571  mm,	Y =   -202.716  mm,	Z =   -247.935  mm,
	W =  90.000 deg,	P =   0.000 deg,	R =   90.000 deg
};
P[1752]{
   GP1:
	UF : 0, UT : 6,		CONFIG : 'N U T, 0, 0, 0',
	X =  187.241  mm,	Y =   -204.185  mm,	Z =   -248.236  mm,
	W =  90.000 deg,	P =   0.000 deg,	R =   90.000 deg
};
P[1753]{
   GP1:
	UF : 0, UT : 6,		CONFIG : 'N U T, 0, 0, 0',
	X =  186.452  mm,	Y =   -204.539  mm,	Z =   -247.989  mm,
	W =  90.000 deg,	P =   0.000 deg,	R =   90.000 deg
};
P[1754]{
   GP1:
	UF : 0, UT : 6,		CONFIG : 'N U T, 0, 0, 0',
	X =  185.519  mm,	Y =   -205.018  mm,	Z =   -247.846  mm,
	W =  90.000 deg,	P =   0.000 deg,	R =   90.000 deg
};
P[1755]{
   GP1:
	UF : 0, UT : 6,		CONFIG : 'N U T, 0, 0, 0',
	X =  184.773  mm,	Y =   -205.574  mm,	Z =   -248.148  mm,
	W =  90.000 deg,	P =   0.000 deg,	R =   90.000 deg
};
P[1756]{
   GP1:
	UF : 0, UT : 6,		CONFIG : 'N U T, 0, 0, 0',
	X =  184.121  mm,	Y =   -205.922  mm,	Z =   -248.079  mm,
	W =  90.000 deg,	P =   0.000 deg,	R =   90.000 deg
};
P[1757]{
   GP1:
	UF : 0, UT : 6,		CONFIG : 'N U T, 0, 0, 0',
	X =  180.900  mm,	Y =   -207.707  mm,	Z =   -247.899  mm,
	W =  90.000 deg,	P =   0.000 deg,	R =   90.000 deg
};
P[1758]{
   GP1:
	UF : 0, UT : 6,		CONFIG : 'N U T, 0, 0, 0',
	X =  179.569  mm,	Y =   -208.584  mm,	Z =   -248.162  mm,
	W =  90.000 deg,	P =   0.000 deg,	R =   90.000 deg
};
P[1759]{
   GP1:
	UF : 0, UT : 6,		CONFIG : 'N U T, 0, 0, 0',
	X =  175.956  mm,	Y =   -210.692  mm,	Z =   -248.214  mm,
	W =  90.000 deg,	P =   0.000 deg,	R =   90.000 deg
};
P[1760]{
   GP1:
	UF : 0, UT : 6,		CONFIG : 'N U T, 0, 0, 0',
	X =  171.838  mm,	Y =   -213.008  mm,	Z =   -248.066  mm,
	W =  90.000 deg,	P =   0.000 deg,	R =   90.000 deg
};
P[1761]{
   GP1:
	UF : 0, UT : 6,		CONFIG : 'N U T, 0, 0, 0',
	X =  171.214  mm,	Y =   -213.377  mm,	Z =   -248.086  mm,
	W =  90.000 deg,	P =   0.000 deg,	R =   90.000 deg
};
P[1762]{
   GP1:
	UF : 0, UT : 6,		CONFIG : 'N U T, 0, 0, 0',
	X =  170.493  mm,	Y =   -213.781  mm,	Z =   -248.054  mm,
	W =  90.000 deg,	P =   0.000 deg,	R =   90.000 deg
};
P[1763]{
   GP1:
	UF : 0, UT : 6,		CONFIG : 'N U T, 0, 0, 0',
	X =  169.192  mm,	Y =   -214.597  mm,	Z =   -248.216  mm,
	W =  90.000 deg,	P =   0.000 deg,	R =   90.000 deg
};
P[1764]{
   GP1:
	UF : 0, UT : 6,		CONFIG : 'N U T, 0, 0, 0',
	X =  163.896  mm,	Y =   -217.604  mm,	Z =   -248.091  mm,
	W =  90.000 deg,	P =   0.000 deg,	R =   90.000 deg
};
P[1765]{
   GP1:
	UF : 0, UT : 6,		CONFIG : 'N U T, 0, 0, 0',
	X =  162.201  mm,	Y =   -218.625  mm,	Z =   -248.193  mm,
	W =  90.000 deg,	P =   0.000 deg,	R =   90.000 deg
};
P[1766]{
   GP1:
	UF : 0, UT : 6,		CONFIG : 'N U T, 0, 0, 0',
	X =  161.060  mm,	Y =   -219.214  mm,	Z =   -248.025  mm,
	W =  90.000 deg,	P =   0.000 deg,	R =   90.000 deg
};
P[1767]{
   GP1:
	UF : 0, UT : 6,		CONFIG : 'N U T, 0, 0, 0',
	X =  158.664  mm,	Y =   -220.660  mm,	Z =   -248.176  mm,
	W =  90.000 deg,	P =   0.000 deg,	R =   90.000 deg
};
P[1768]{
   GP1:
	UF : 0, UT : 6,		CONFIG : 'N U T, 0, 0, 0',
	X =  156.586  mm,	Y =   -221.830  mm,	Z =   -248.103  mm,
	W =  90.000 deg,	P =   0.000 deg,	R =   90.000 deg
};
P[1769]{
   GP1:
	UF : 0, UT : 6,		CONFIG : 'N U T, 0, 0, 0',
	X =  155.220  mm,	Y =   -222.598  mm,	Z =   -248.052  mm,
	W =  90.000 deg,	P =   0.000 deg,	R =   90.000 deg
};
P[1770]{
   GP1:
	UF : 0, UT : 6,		CONFIG : 'N U T, 0, 0, 0',
	X =  154.063  mm,	Y =   -223.324  mm,	Z =   -248.191  mm,
	W =  90.000 deg,	P =   0.000 deg,	R =   90.000 deg
};
P[1771]{
   GP1:
	UF : 0, UT : 6,		CONFIG : 'N U T, 0, 0, 0',
	X =  152.597  mm,	Y =   -224.100  mm,	Z =   -248.021  mm,
	W =  90.000 deg,	P =   0.000 deg,	R =   90.000 deg
};
P[1772]{
   GP1:
	UF : 0, UT : 6,		CONFIG : 'N U T, 0, 0, 0',
	X =  151.470  mm,	Y =   -224.828  mm,	Z =   -248.210  mm,
	W =  90.000 deg,	P =   0.000 deg,	R =   90.000 deg
};
P[1773]{
   GP1:
	UF : 0, UT : 6,		CONFIG : 'N U T, 0, 0, 0',
	X =  147.560  mm,	Y =   -227.088  mm,	Z =   -248.216  mm,
	W =  90.000 deg,	P =   0.000 deg,	R =   90.000 deg
};
P[1774]{
   GP1:
	UF : 0, UT : 6,		CONFIG : 'N U T, 0, 0, 0',
	X =  146.858  mm,	Y =   -227.458  mm,	Z =   -248.131  mm,
	W =  90.000 deg,	P =   0.000 deg,	R =   90.000 deg
};
P[1775]{
   GP1:
	UF : 0, UT : 6,		CONFIG : 'N U T, 0, 0, 0',
	X =  145.866  mm,	Y =   -228.012  mm,	Z =   -248.087  mm,
	W =  90.000 deg,	P =   0.000 deg,	R =   90.000 deg
};
P[1776]{
   GP1:
	UF : 0, UT : 6,		CONFIG : 'N U T, 0, 0, 0',
	X =  144.720  mm,	Y =   -228.599  mm,	Z =   -247.904  mm,
	W =  90.000 deg,	P =   0.000 deg,	R =   90.000 deg
};
P[1777]{
   GP1:
	UF : 0, UT : 6,		CONFIG : 'N U T, 0, 0, 0',
	X =  143.466  mm,	Y =   -229.366  mm,	Z =   -248.007  mm,
	W =  90.000 deg,	P =   0.000 deg,	R =   90.000 deg
};
P[1778]{
   GP1:
	UF : 0, UT : 6,		CONFIG : 'N U T, 0, 0, 0',
	X =  142.551  mm,	Y =   -229.931  mm,	Z =   -248.097  mm,
	W =  90.000 deg,	P =   0.000 deg,	R =   90.000 deg
};
P[1779]{
   GP1:
	UF : 0, UT : 6,		CONFIG : 'N U T, 0, 0, 0',
	X =  140.718  mm,	Y =   -231.042  mm,	Z =   -248.225  mm,
	W =  90.000 deg,	P =   0.000 deg,	R =   90.000 deg
};
P[1780]{
   GP1:
	UF : 0, UT : 6,		CONFIG : 'N U T, 0, 0, 0',
	X =  139.767  mm,	Y =   -231.421  mm,	Z =   -247.812  mm,
	W =  90.000 deg,	P =   0.000 deg,	R =   90.000 deg
};
P[1781]{
   GP1:
	UF : 0, UT : 6,		CONFIG : 'N U T, 0, 0, 0',
	X =  138.577  mm,	Y =   -232.117  mm,	Z =   -247.834  mm,
	W =  90.000 deg,	P =   0.000 deg,	R =   90.000 deg
};
P[1782]{
   GP1:
	UF : 0, UT : 6,		CONFIG : 'N U T, 0, 0, 0',
	X =  136.612  mm,	Y =   -233.422  mm,	Z =   -248.248  mm,
	W =  90.000 deg,	P =   0.000 deg,	R =   90.000 deg
};
P[1783]{
   GP1:
	UF : 0, UT : 6,		CONFIG : 'N U T, 0, 0, 0',
	X =  135.655  mm,	Y =   -233.957  mm,	Z =   -248.205  mm,
	W =  90.000 deg,	P =   0.000 deg,	R =   90.000 deg
};
P[1784]{
   GP1:
	UF : 0, UT : 6,		CONFIG : 'N U T, 0, 0, 0',
	X =  134.528  mm,	Y =   -234.433  mm,	Z =   -247.779  mm,
	W =  90.000 deg,	P =   0.000 deg,	R =   90.000 deg
};
P[1785]{
   GP1:
	UF : 0, UT : 6,		CONFIG : 'N U T, 0, 0, 0',
	X =  132.974  mm,	Y =   -235.413  mm,	Z =   -247.978  mm,
	W =  90.000 deg,	P =   0.000 deg,	R =   90.000 deg
};
P[1786]{
   GP1:
	UF : 0, UT : 6,		CONFIG : 'N U T, 0, 0, 0',
	X =  131.454  mm,	Y =   -236.317  mm,	Z =   -248.045  mm,
	W =  90.000 deg,	P =   0.000 deg,	R =   90.000 deg
};
P[1787]{
   GP1:
	UF : 0, UT : 6,		CONFIG : 'N U T, 0, 0, 0',
	X =  129.608  mm,	Y =   -237.336  mm,	Z =   -247.932  mm,
	W =  90.000 deg,	P =   0.000 deg,	R =   90.000 deg
};
P[1788]{
   GP1:
	UF : 0, UT : 6,		CONFIG : 'N U T, 0, 0, 0',
	X =  128.456  mm,	Y =   -237.997  mm,	Z =   -247.922  mm,
	W =  90.000 deg,	P =   0.000 deg,	R =   90.000 deg
};
P[1789]{
   GP1:
	UF : 0, UT : 6,		CONFIG : 'N U T, 0, 0, 0',
	X =  127.638  mm,	Y =   -238.508  mm,	Z =   -248.013  mm,
	W =  90.000 deg,	P =   0.000 deg,	R =   90.000 deg
};
P[1790]{
   GP1:
	UF : 0, UT : 6,		CONFIG : 'N U T, 0, 0, 0',
	X =  123.726  mm,	Y =   -240.729  mm,	Z =   -247.924  mm,
	W =  90.000 deg,	P =   0.000 deg,	R =   90.000 deg
};
P[1791]{
   GP1:
	UF : 0, UT : 6,		CONFIG : 'N U T, 0, 0, 0',
	X =  121.664  mm,	Y =   -241.957  mm,	Z =   -248.015  mm,
	W =  90.000 deg,	P =   0.000 deg,	R =   90.000 deg
};
P[1792]{
   GP1:
	UF : 0, UT : 6,		CONFIG : 'N U T, 0, 0, 0',
	X =  120.580  mm,	Y =   -242.494  mm,	Z =   -247.797  mm,
	W =  90.000 deg,	P =   0.000 deg,	R =   90.000 deg
};
P[1793]{
   GP1:
	UF : 0, UT : 6,		CONFIG : 'N U T, 0, 0, 0',
	X =  117.690  mm,	Y =   -244.185  mm,	Z =   -247.853  mm,
	W =  90.000 deg,	P =   0.000 deg,	R =   90.000 deg
};
P[1794]{
   GP1:
	UF : 0, UT : 6,		CONFIG : 'N U T, 0, 0, 0',
	X =  115.373  mm,	Y =   -245.533  mm,	Z =   -247.876  mm,
	W =  90.000 deg,	P =   0.000 deg,	R =   90.000 deg
};
P[1795]{
   GP1:
	UF : 0, UT : 6,		CONFIG : 'N U T, 0, 0, 0',
	X =  113.686  mm,	Y =   -246.619  mm,	Z =   -248.148  mm,
	W =  90.000 deg,	P =   0.000 deg,	R =   90.000 deg
};
P[1796]{
   GP1:
	UF : 0, UT : 6,		CONFIG : 'N U T, 0, 0, 0',
	X =  112.989  mm,	Y =   -246.944  mm,	Z =   -247.961  mm,
	W =  90.000 deg,	P =   0.000 deg,	R =   90.000 deg
};
P[1797]{
   GP1:
	UF : 0, UT : 6,		CONFIG : 'N U T, 0, 0, 0',
	X =  111.975  mm,	Y =   -247.507  mm,	Z =   -247.908  mm,
	W =  90.000 deg,	P =   0.000 deg,	R =   90.000 deg
};
P[1798]{
   GP1:
	UF : 0, UT : 6,		CONFIG : 'N U T, 0, 0, 0',
	X =  110.986  mm,	Y =   -248.046  mm,	Z =   -247.828  mm,
	W =  90.000 deg,	P =   0.000 deg,	R =   90.000 deg
};
P[1799]{
   GP1:
	UF : 0, UT : 6,		CONFIG : 'N U T, 0, 0, 0',
	X =  109.707  mm,	Y =   -248.883  mm,	Z =   -248.069  mm,
	W =  90.000 deg,	P =   0.000 deg,	R =   90.000 deg
};
P[1800]{
   GP1:
	UF : 0, UT : 6,		CONFIG : 'N U T, 0, 0, 0',
	X =  108.347  mm,	Y =   -249.635  mm,	Z =   -247.988  mm,
	W =  90.000 deg,	P =   0.000 deg,	R =   90.000 deg
};
P[1801]{
   GP1:
	UF : 0, UT : 6,		CONFIG : 'N U T, 0, 0, 0',
	X =  105.962  mm,	Y =   -251.099  mm,	Z =   -248.199  mm,
	W =  90.000 deg,	P =   0.000 deg,	R =   90.000 deg
};
P[1802]{
   GP1:
	UF : 0, UT : 6,		CONFIG : 'N U T, 0, 0, 0',
	X =  105.202  mm,	Y =   -251.547  mm,	Z =   -248.219  mm,
	W =  90.000 deg,	P =   0.000 deg,	R =   90.000 deg
};
P[1803]{
   GP1:
	UF : 0, UT : 6,		CONFIG : 'N U T, 0, 0, 0',
	X =  104.062  mm,	Y =   -252.107  mm,	Z =   -247.981  mm,
	W =  90.000 deg,	P =   0.000 deg,	R =   90.000 deg
};
P[1804]{
   GP1:
	UF : 0, UT : 6,		CONFIG : 'N U T, 0, 0, 0',
	X =  102.478  mm,	Y =   -250.670  mm,	Z =   -242.275  mm,
	W =  90.000 deg,	P =   0.000 deg,	R =   90.000 deg
};
P[1805]{
   GP1:
	UF : 0, UT : 6,		CONFIG : 'N U T, 0, 0, 0',
	X =  101.193  mm,	Y =   -251.368  mm,	Z =   -242.167  mm,
	W =  90.000 deg,	P =   0.000 deg,	R =   90.000 deg
};
P[1806]{
   GP1:
	UF : 0, UT : 6,		CONFIG : 'N U T, 0, 0, 0',
	X =  97.386  mm,	Y =   -253.593  mm,	Z =   -242.233  mm,
	W =  90.000 deg,	P =   0.000 deg,	R =   90.000 deg
};
P[1807]{
   GP1:
	UF : 0, UT : 6,		CONFIG : 'N U T, 0, 0, 0',
	X =  96.420  mm,	Y =   -254.177  mm,	Z =   -242.294  mm,
	W =  90.000 deg,	P =   0.000 deg,	R =   90.000 deg
};
P[1808]{
   GP1:
	UF : 0, UT : 6,		CONFIG : 'N U T, 0, 0, 0',
	X =  94.579  mm,	Y =   -255.099  mm,	Z =   -241.955  mm,
	W =  90.000 deg,	P =   0.000 deg,	R =   90.000 deg
};
P[1809]{
   GP1:
	UF : 0, UT : 6,		CONFIG : 'N U T, 0, 0, 0',
	X =  94.014  mm,	Y =   -255.546  mm,	Z =   -242.248  mm,
	W =  90.000 deg,	P =   0.000 deg,	R =   90.000 deg
};
P[1810]{
   GP1:
	UF : 0, UT : 6,		CONFIG : 'N U T, 0, 0, 0',
	X =  92.688  mm,	Y =   -256.257  mm,	Z =   -242.116  mm,
	W =  90.000 deg,	P =   0.000 deg,	R =   90.000 deg
};
P[1811]{
   GP1:
	UF : 0, UT : 6,		CONFIG : 'N U T, 0, 0, 0',
	X =  91.989  mm,	Y =   -256.700  mm,	Z =   -242.212  mm,
	W =  90.000 deg,	P =   0.000 deg,	R =   90.000 deg
};
P[1812]{
   GP1:
	UF : 0, UT : 6,		CONFIG : 'N U T, 0, 0, 0',
	X =  91.138  mm,	Y =   -257.220  mm,	Z =   -242.280  mm,
	W =  90.000 deg,	P =   0.000 deg,	R =   90.000 deg
};
P[1813]{
   GP1:
	UF : 0, UT : 6,		CONFIG : 'N U T, 0, 0, 0',
	X =  90.007  mm,	Y =   -257.900  mm,	Z =   -242.346  mm,
	W =  90.000 deg,	P =   0.000 deg,	R =   90.000 deg
};
P[1814]{
   GP1:
	UF : 0, UT : 6,		CONFIG : 'N U T, 0, 0, 0',
	X =  89.048  mm,	Y =   -258.449  mm,	Z =   -242.334  mm,
	W =  90.000 deg,	P =   0.000 deg,	R =   90.000 deg
};
P[1815]{
   GP1:
	UF : 0, UT : 6,		CONFIG : 'N U T, 0, 0, 0',
	X =  78.196  mm,	Y =   -264.569  mm,	Z =   -241.981  mm,
	W =  90.000 deg,	P =   0.000 deg,	R =   90.000 deg
};
P[1816]{
   GP1:
	UF : 0, UT : 6,		CONFIG : 'N U T, 0, 0, 0',
	X =  75.324  mm,	Y =   -266.361  mm,	Z =   -242.303  mm,
	W =  90.000 deg,	P =   0.000 deg,	R =   90.000 deg
};
P[1817]{
   GP1:
	UF : 0, UT : 6,		CONFIG : 'N U T, 0, 0, 0',
	X =  74.280  mm,	Y =   -266.937  mm,	Z =   -242.240  mm,
	W =  90.000 deg,	P =   0.000 deg,	R =   90.000 deg
};
P[1818]{
   GP1:
	UF : 0, UT : 6,		CONFIG : 'N U T, 0, 0, 0',
	X =  72.171  mm,	Y =   -268.135  mm,	Z =   -242.194  mm,
	W =  90.000 deg,	P =   0.000 deg,	R =   90.000 deg
};
P[1819]{
   GP1:
	UF : 0, UT : 6,		CONFIG : 'N U T, 0, 0, 0',
	X =  70.786  mm,	Y =   -268.829  mm,	Z =   -241.933  mm,
	W =  90.000 deg,	P =   0.000 deg,	R =   90.000 deg
};
P[1820]{
   GP1:
	UF : 0, UT : 6,		CONFIG : 'N U T, 0, 0, 0',
	X =  66.999  mm,	Y =   -271.157  mm,	Z =   -242.279  mm,
	W =  90.000 deg,	P =   0.000 deg,	R =   90.000 deg
};
P[1821]{
   GP1:
	UF : 0, UT : 6,		CONFIG : 'N U T, 0, 0, 0',
	X =  66.157  mm,	Y =   -271.604  mm,	Z =   -242.184  mm,
	W =  90.000 deg,	P =   0.000 deg,	R =   90.000 deg
};
P[1822]{
   GP1:
	UF : 0, UT : 6,		CONFIG : 'N U T, 0, 0, 0',
	X =  63.185  mm,	Y =   -273.302  mm,	Z =   -242.140  mm,
	W =  90.000 deg,	P =   0.000 deg,	R =   90.000 deg
};
P[1823]{
   GP1:
	UF : 0, UT : 6,		CONFIG : 'N U T, 0, 0, 0',
	X =  61.397  mm,	Y =   -274.378  mm,	Z =   -242.246  mm,
	W =  90.000 deg,	P =   0.000 deg,	R =   90.000 deg
};
P[1824]{
   GP1:
	UF : 0, UT : 6,		CONFIG : 'N U T, 0, 0, 0',
	X =  60.357  mm,	Y =   -274.865  mm,	Z =   -241.970  mm,
	W =  90.000 deg,	P =   0.000 deg,	R =   90.000 deg
};
P[1825]{
   GP1:
	UF : 0, UT : 6,		CONFIG : 'N U T, 0, 0, 0',
	X =  59.166  mm,	Y =   -275.629  mm,	Z =   -242.157  mm,
	W =  90.000 deg,	P =   0.000 deg,	R =   90.000 deg
};
P[1826]{
   GP1:
	UF : 0, UT : 6,		CONFIG : 'N U T, 0, 0, 0',
	X =  58.386  mm,	Y =   -276.153  mm,	Z =   -242.335  mm,
	W =  90.000 deg,	P =   0.000 deg,	R =   90.000 deg
};
P[1827]{
   GP1:
	UF : 0, UT : 6,		CONFIG : 'N U T, 0, 0, 0',
	X =  56.071  mm,	Y =   -277.487  mm,	Z =   -242.328  mm,
	W =  90.000 deg,	P =   0.000 deg,	R =   90.000 deg
};
P[1828]{
   GP1:
	UF : 0, UT : 6,		CONFIG : 'N U T, 0, 0, 0',
	X =  54.156  mm,	Y =   -278.560  mm,	Z =   -242.248  mm,
	W =  90.000 deg,	P =   0.000 deg,	R =   90.000 deg
};
P[1829]{
   GP1:
	UF : 0, UT : 6,		CONFIG : 'N U T, 0, 0, 0',
	X =  52.969  mm,	Y =   -279.248  mm,	Z =   -242.254  mm,
	W =  90.000 deg,	P =   0.000 deg,	R =   90.000 deg
};
P[1830]{
   GP1:
	UF : 0, UT : 6,		CONFIG : 'N U T, 0, 0, 0',
	X =  51.438  mm,	Y =   -279.990  mm,	Z =   -241.909  mm,
	W =  90.000 deg,	P =   0.000 deg,	R =   90.000 deg
};
P[1831]{
   GP1:
	UF : 0, UT : 6,		CONFIG : 'N U T, 0, 0, 0',
	X =  50.777  mm,	Y =   -280.449  mm,	Z =   -242.100  mm,
	W =  90.000 deg,	P =   0.000 deg,	R =   90.000 deg
};
P[1832]{
   GP1:
	UF : 0, UT : 6,		CONFIG : 'N U T, 0, 0, 0',
	X =  48.869  mm,	Y =   -281.668  mm,	Z =   -242.383  mm,
	W =  90.000 deg,	P =   0.000 deg,	R =   90.000 deg
};
P[1833]{
   GP1:
	UF : 0, UT : 6,		CONFIG : 'N U T, 0, 0, 0',
	X =  47.876  mm,	Y =   -282.215  mm,	Z =   -242.318  mm,
	W =  90.000 deg,	P =   0.000 deg,	R =   90.000 deg
};
P[1834]{
   GP1:
	UF : 0, UT : 6,		CONFIG : 'N U T, 0, 0, 0',
	X =  46.563  mm,	Y =   -282.903  mm,	Z =   -242.149  mm,
	W =  90.000 deg,	P =   0.000 deg,	R =   90.000 deg
};
P[1835]{
   GP1:
	UF : 0, UT : 6,		CONFIG : 'N U T, 0, 0, 0',
	X =  44.597  mm,	Y =   -284.041  mm,	Z =   -242.156  mm,
	W =  90.000 deg,	P =   0.000 deg,	R =   90.000 deg
};
P[1836]{
   GP1:
	UF : 0, UT : 6,		CONFIG : 'N U T, 0, 0, 0',
	X =  41.853  mm,	Y =   -285.696  mm,	Z =   -242.327  mm,
	W =  90.000 deg,	P =   0.000 deg,	R =   90.000 deg
};
P[1837]{
   GP1:
	UF : 0, UT : 6,		CONFIG : 'N U T, 0, 0, 0',
	X =  40.046  mm,	Y =   -286.626  mm,	Z =   -242.052  mm,
	W =  90.000 deg,	P =   0.000 deg,	R =   90.000 deg
};
P[1838]{
   GP1:
	UF : 0, UT : 6,		CONFIG : 'N U T, 0, 0, 0',
	X =  38.871  mm,	Y =   -287.330  mm,	Z =   -242.114  mm,
	W =  90.000 deg,	P =   0.000 deg,	R =   90.000 deg
};
P[1839]{
   GP1:
	UF : 0, UT : 6,		CONFIG : 'N U T, 0, 0, 0',
	X =  37.847  mm,	Y =   -287.971  mm,	Z =   -242.232  mm,
	W =  90.000 deg,	P =   0.000 deg,	R =   90.000 deg
};
P[1840]{
   GP1:
	UF : 0, UT : 6,		CONFIG : 'N U T, 0, 0, 0',
	X =  34.731  mm,	Y =   -289.832  mm,	Z =   -242.384  mm,
	W =  90.000 deg,	P =   0.000 deg,	R =   90.000 deg
};
P[1841]{
   GP1:
	UF : 0, UT : 6,		CONFIG : 'N U T, 0, 0, 0',
	X =  34.079  mm,	Y =   -290.138  mm,	Z =   -242.213  mm,
	W =  90.000 deg,	P =   0.000 deg,	R =   90.000 deg
};
P[1842]{
   GP1:
	UF : 0, UT : 6,		CONFIG : 'N U T, 0, 0, 0',
	X =  31.958  mm,	Y =   -291.416  mm,	Z =   -242.344  mm,
	W =  90.000 deg,	P =   0.000 deg,	R =   90.000 deg
};
P[1843]{
   GP1:
	UF : 0, UT : 6,		CONFIG : 'N U T, 0, 0, 0',
	X =  27.744  mm,	Y =   -293.759  mm,	Z =   -242.123  mm,
	W =  90.000 deg,	P =   0.000 deg,	R =   90.000 deg
};
P[1844]{
   GP1:
	UF : 0, UT : 6,		CONFIG : 'N U T, 0, 0, 0',
	X =  26.741  mm,	Y =   -294.338  mm,	Z =   -242.123  mm,
	W =  90.000 deg,	P =   0.000 deg,	R =   90.000 deg
};
P[1845]{
   GP1:
	UF : 0, UT : 6,		CONFIG : 'N U T, 0, 0, 0',
	X =  20.191  mm,	Y =   -298.113  mm,	Z =   -242.107  mm,
	W =  90.000 deg,	P =   0.000 deg,	R =   90.000 deg
};
P[1846]{
   GP1:
	UF : 0, UT : 6,		CONFIG : 'N U T, 0, 0, 0',
	X =  19.352  mm,	Y =   -298.613  mm,	Z =   -242.146  mm,
	W =  90.000 deg,	P =   0.000 deg,	R =   90.000 deg
};
P[1847]{
   GP1:
	UF : 0, UT : 6,		CONFIG : 'N U T, 0, 0, 0',
	X =  8.205  mm,	Y =   -304.977  mm,	Z =   -241.971  mm,
	W =  90.000 deg,	P =   0.000 deg,	R =   90.000 deg
};
P[1848]{
   GP1:
	UF : 0, UT : 6,		CONFIG : 'N U T, 0, 0, 0',
	X =  5.825  mm,	Y =   -306.493  mm,	Z =   -242.314  mm,
	W =  90.000 deg,	P =   0.000 deg,	R =   90.000 deg
};
P[1849]{
   GP1:
	UF : 0, UT : 6,		CONFIG : 'N U T, 0, 0, 0',
	X =  2.381  mm,	Y =   -308.489  mm,	Z =   -242.332  mm,
	W =  90.000 deg,	P =   0.000 deg,	R =   90.000 deg
};
P[1850]{
   GP1:
	UF : 0, UT : 6,		CONFIG : 'N U T, 0, 0, 0',
	X =  1.457  mm,	Y =   -308.861  mm,	Z =   -241.940  mm,
	W =  90.000 deg,	P =   0.000 deg,	R =   90.000 deg
};
P[1851]{
   GP1:
	UF : 0, UT : 6,		CONFIG : 'N U T, 0, 0, 0',
	X =  0.645  mm,	Y =   -309.409  mm,	Z =   -242.131  mm,
	W =  90.000 deg,	P =   0.000 deg,	R =   90.000 deg
};
P[1852]{
   GP1:
	UF : 0, UT : 6,		CONFIG : 'N U T, 0, 0, 0',
	X =  -0.039  mm,	Y =   -309.903  mm,	Z =   -242.373  mm,
	W =  90.000 deg,	P =   0.000 deg,	R =   90.000 deg
};
P[1853]{
   GP1:
	UF : 0, UT : 6,		CONFIG : 'N U T, 0, 0, 0',
	X =  -2.871  mm,	Y =   -311.382  mm,	Z =   -241.993  mm,
	W =  90.000 deg,	P =   0.000 deg,	R =   90.000 deg
};
P[1854]{
   GP1:
	UF : 0, UT : 6,		CONFIG : 'N U T, 0, 0, 0',
	X =  -3.631  mm,	Y =   -311.920  mm,	Z =   -242.234  mm,
	W =  90.000 deg,	P =   0.000 deg,	R =   90.000 deg
};
P[1855]{
   GP1:
	UF : 0, UT : 6,		CONFIG : 'N U T, 0, 0, 0',
	X =  -5.894  mm,	Y =   -313.248  mm,	Z =   -242.284  mm,
	W =  90.000 deg,	P =   0.000 deg,	R =   90.000 deg
};
P[1856]{
   GP1:
	UF : 0, UT : 6,		CONFIG : 'N U T, 0, 0, 0',
	X =  -14.582  mm,	Y =   -318.147  mm,	Z =   -242.000  mm,
	W =  90.000 deg,	P =   0.000 deg,	R =   90.000 deg
};
P[1857]{
   GP1:
	UF : 0, UT : 6,		CONFIG : 'N U T, 0, 0, 0',
	X =  -16.008  mm,	Y =   -319.062  mm,	Z =   -242.226  mm,
	W =  90.000 deg,	P =   0.000 deg,	R =   90.000 deg
};
P[1858]{
   GP1:
	UF : 0, UT : 6,		CONFIG : 'N U T, 0, 0, 0',
	X =  -18.600  mm,	Y =   -320.606  mm,	Z =   -242.341  mm,
	W =  90.000 deg,	P =   0.000 deg,	R =   90.000 deg
};
P[1859]{
   GP1:
	UF : 0, UT : 6,		CONFIG : 'N U T, 0, 0, 0',
	X =  -21.539  mm,	Y =   -322.169  mm,	Z =   -242.014  mm,
	W =  90.000 deg,	P =   0.000 deg,	R =   90.000 deg
};
P[1860]{
   GP1:
	UF : 0, UT : 6,		CONFIG : 'N U T, 0, 0, 0',
	X =  -25.350  mm,	Y =   -324.487  mm,	Z =   -242.299  mm,
	W =  90.000 deg,	P =   0.000 deg,	R =   90.000 deg
};
P[1861]{
   GP1:
	UF : 0, UT : 6,		CONFIG : 'N U T, 0, 0, 0',
	X =  -27.281  mm,	Y =   -325.637  mm,	Z =   -242.385  mm,
	W =  90.000 deg,	P =   0.000 deg,	R =   90.000 deg
};
P[1862]{
   GP1:
	UF : 0, UT : 6,		CONFIG : 'N U T, 0, 0, 0',
	X =  -28.898  mm,	Y =   -326.407  mm,	Z =   -241.986  mm,
	W =  90.000 deg,	P =   0.000 deg,	R =   90.000 deg
};
P[1863]{
   GP1:
	UF : 0, UT : 6,		CONFIG : 'N U T, 0, 0, 0',
	X =  -29.668  mm,	Y =   -327.001  mm,	Z =   -242.349  mm,
	W =  90.000 deg,	P =   0.000 deg,	R =   90.000 deg
};
P[1864]{
   GP1:
	UF : 0, UT : 6,		CONFIG : 'N U T, 0, 0, 0',
	X =  -30.744  mm,	Y =   -327.489  mm,	Z =   -242.027  mm,
	W =  90.000 deg,	P =   0.000 deg,	R =   90.000 deg
};
P[1865]{
   GP1:
	UF : 0, UT : 6,		CONFIG : 'N U T, 0, 0, 0',
	X =  -31.379  mm,	Y =   -327.918  mm,	Z =   -242.177  mm,
	W =  90.000 deg,	P =   0.000 deg,	R =   90.000 deg
};
P[1866]{
   GP1:
	UF : 0, UT : 6,		CONFIG : 'N U T, 0, 0, 0',
	X =  -34.853  mm,	Y =   -329.965  mm,	Z =   -242.279  mm,
	W =  90.000 deg,	P =   0.000 deg,	R =   90.000 deg
};
P[1867]{
   GP1:
	UF : 0, UT : 6,		CONFIG : 'N U T, 0, 0, 0',
	X =  -37.787  mm,	Y =   -331.547  mm,	Z =   -242.006  mm,
	W =  90.000 deg,	P =   0.000 deg,	R =   90.000 deg
};
P[1868]{
   GP1:
	UF : 0, UT : 6,		CONFIG : 'N U T, 0, 0, 0',
	X =  -38.247  mm,	Y =   -331.925  mm,	Z =   -242.276  mm,
	W =  90.000 deg,	P =   0.000 deg,	R =   90.000 deg
};
P[1869]{
   GP1:
	UF : 0, UT : 6,		CONFIG : 'N U T, 0, 0, 0',
	X =  -42.498  mm,	Y =   -334.400  mm,	Z =   -242.328  mm,
	W =  90.000 deg,	P =   0.000 deg,	R =   90.000 deg
};
P[1870]{
   GP1:
	UF : 0, UT : 6,		CONFIG : 'N U T, 0, 0, 0',
	X =  -43.122  mm,	Y =   -334.638  mm,	Z =   -242.031  mm,
	W =  90.000 deg,	P =   0.000 deg,	R =   90.000 deg
};
P[1871]{
   GP1:
	UF : 0, UT : 6,		CONFIG : 'N U T, 0, 0, 0',
	X =  -44.230  mm,	Y =   -335.226  mm,	Z =   -241.908  mm,
	W =  90.000 deg,	P =   0.000 deg,	R =   90.000 deg
};
P[1872]{
   GP1:
	UF : 0, UT : 6,		CONFIG : 'N U T, 0, 0, 0',
	X =  -44.807  mm,	Y =   -335.610  mm,	Z =   -242.029  mm,
	W =  90.000 deg,	P =   0.000 deg,	R =   90.000 deg
};
P[1873]{
   GP1:
	UF : 0, UT : 6,		CONFIG : 'N U T, 0, 0, 0',
	X =  -45.956  mm,	Y =   -336.388  mm,	Z =   -242.307  mm,
	W =  90.000 deg,	P =   0.000 deg,	R =   90.000 deg
};
P[1874]{
   GP1:
	UF : 0, UT : 6,		CONFIG : 'N U T, 0, 0, 0',
	X =  -49.438  mm,	Y =   -338.420  mm,	Z =   -242.361  mm,
	W =  90.000 deg,	P =   0.000 deg,	R =   90.000 deg
};
P[1875]{
   GP1:
	UF : 0, UT : 6,		CONFIG : 'N U T, 0, 0, 0',
	X =  -51.548  mm,	Y =   -339.599  mm,	Z =   -242.263  mm,
	W =  90.000 deg,	P =   0.000 deg,	R =   90.000 deg
};
P[1876]{
   GP1:
	UF : 0, UT : 6,		CONFIG : 'N U T, 0, 0, 0',
	X =  -55.904  mm,	Y =   -342.045  mm,	Z =   -242.096  mm,
	W =  90.000 deg,	P =   0.000 deg,	R =   90.000 deg
};
P[1877]{
   GP1:
	UF : 0, UT : 6,		CONFIG : 'N U T, 0, 0, 0',
	X =  -57.598  mm,	Y =   -343.025  mm,	Z =   -242.102  mm,
	W =  90.000 deg,	P =   0.000 deg,	R =   90.000 deg
};
P[1878]{
   GP1:
	UF : 0, UT : 6,		CONFIG : 'N U T, 0, 0, 0',
	X =  -60.027  mm,	Y =   -344.449  mm,	Z =   -242.155  mm,
	W =  90.000 deg,	P =   0.000 deg,	R =   90.000 deg
};
P[1879]{
   GP1:
	UF : 0, UT : 6,		CONFIG : 'N U T, 0, 0, 0',
	X =  -60.814  mm,	Y =   -344.928  mm,	Z =   -242.215  mm,
	W =  90.000 deg,	P =   0.000 deg,	R =   90.000 deg
};
P[1880]{
   GP1:
	UF : 0, UT : 6,		CONFIG : 'N U T, 0, 0, 0',
	X =  -62.757  mm,	Y =   -346.061  mm,	Z =   -242.239  mm,
	W =  90.000 deg,	P =   0.000 deg,	R =   90.000 deg
};
P[1881]{
   GP1:
	UF : 0, UT : 6,		CONFIG : 'N U T, 0, 0, 0',
	X =  -65.492  mm,	Y =   -347.568  mm,	Z =   -242.063  mm,
	W =  90.000 deg,	P =   0.000 deg,	R =   90.000 deg
};
P[1882]{
   GP1:
	UF : 0, UT : 6,		CONFIG : 'N U T, 0, 0, 0',
	X =  -66.970  mm,	Y =   -348.400  mm,	Z =   -242.012  mm,
	W =  90.000 deg,	P =   0.000 deg,	R =   90.000 deg
};
P[1883]{
   GP1:
	UF : 0, UT : 6,		CONFIG : 'N U T, 0, 0, 0',
	X =  -68.647  mm,	Y =   -349.452  mm,	Z =   -242.216  mm,
	W =  90.000 deg,	P =   0.000 deg,	R =   90.000 deg
};
P[1884]{
   GP1:
	UF : 0, UT : 6,		CONFIG : 'N U T, 0, 0, 0',
	X =  -69.611  mm,	Y =   -349.944  mm,	Z =   -242.061  mm,
	W =  90.000 deg,	P =   0.000 deg,	R =   90.000 deg
};
P[1885]{
   GP1:
	UF : 0, UT : 6,		CONFIG : 'N U T, 0, 0, 0',
	X =  -72.352  mm,	Y =   -351.597  mm,	Z =   -242.228  mm,
	W =  90.000 deg,	P =   0.000 deg,	R =   90.000 deg
};
P[1886]{
   GP1:
	UF : 0, UT : 6,		CONFIG : 'N U T, 0, 0, 0',
	X =  -76.561  mm,	Y =   -354.017  mm,	Z =   -242.205  mm,
	W =  90.000 deg,	P =   0.000 deg,	R =   90.000 deg
};
P[1887]{
   GP1:
	UF : 0, UT : 6,		CONFIG : 'N U T, 0, 0, 0',
	X =  -77.161  mm,	Y =   -354.352  mm,	Z =   -242.174  mm,
	W =  90.000 deg,	P =   0.000 deg,	R =   90.000 deg
};
P[1888]{
   GP1:
	UF : 0, UT : 6,		CONFIG : 'N U T, 0, 0, 0',
	X =  -81.003  mm,	Y =   -356.656  mm,	Z =   -242.383  mm,
	W =  90.000 deg,	P =   0.000 deg,	R =   90.000 deg
};
P[1889]{
   GP1:
	UF : 0, UT : 6,		CONFIG : 'N U T, 0, 0, 0',
	X =  -83.128  mm,	Y =   -357.834  mm,	Z =   -242.266  mm,
	W =  90.000 deg,	P =   0.000 deg,	R =   90.000 deg
};
P[1890]{
   GP1:
	UF : 0, UT : 6,		CONFIG : 'N U T, 0, 0, 0',
	X =  -86.437  mm,	Y =   -359.615  mm,	Z =   -241.955  mm,
	W =  90.000 deg,	P =   0.000 deg,	R =   90.000 deg
};
P[1891]{
   GP1:
	UF : 0, UT : 6,		CONFIG : 'N U T, 0, 0, 0',
	X =  -87.174  mm,	Y =   -360.061  mm,	Z =   -242.004  mm,
	W =  90.000 deg,	P =   0.000 deg,	R =   90.000 deg
};
P[1892]{
   GP1:
	UF : 0, UT : 6,		CONFIG : 'N U T, 0, 0, 0',
	X =  -90.784  mm,	Y =   -362.214  mm,	Z =   -242.167  mm,
	W =  90.000 deg,	P =   0.000 deg,	R =   90.000 deg
};
P[1893]{
   GP1:
	UF : 0, UT : 6,		CONFIG : 'N U T, 0, 0, 0',
	X =  -91.770  mm,	Y =   -362.722  mm,	Z =   -242.021  mm,
	W =  90.000 deg,	P =   0.000 deg,	R =   90.000 deg
};
P[1894]{
   GP1:
	UF : 0, UT : 6,		CONFIG : 'N U T, 0, 0, 0',
	X =  -93.342  mm,	Y =   -363.752  mm,	Z =   -242.316  mm,
	W =  90.000 deg,	P =   0.000 deg,	R =   90.000 deg
};
P[1895]{
   GP1:
	UF : 0, UT : 6,		CONFIG : 'N U T, 0, 0, 0',
	X =  -94.228  mm,	Y =   -364.190  mm,	Z =   -242.139  mm,
	W =  90.000 deg,	P =   0.000 deg,	R =   90.000 deg
};
P[1896]{
   GP1:
	UF : 0, UT : 6,		CONFIG : 'N U T, 0, 0, 0',
	X =  -95.860  mm,	Y =   -365.165  mm,	Z =   -242.216  mm,
	W =  90.000 deg,	P =   0.000 deg,	R =   90.000 deg
};
P[1897]{
   GP1:
	UF : 0, UT : 6,		CONFIG : 'N U T, 0, 0, 0',
	X =  -97.501  mm,	Y =   -366.090  mm,	Z =   -242.161  mm,
	W =  90.000 deg,	P =   0.000 deg,	R =   90.000 deg
};
P[1898]{
   GP1:
	UF : 0, UT : 6,		CONFIG : 'N U T, 0, 0, 0',
	X =  -98.358  mm,	Y =   -366.626  mm,	Z =   -242.264  mm,
	W =  90.000 deg,	P =   0.000 deg,	R =   90.000 deg
};
P[1899]{
   GP1:
	UF : 0, UT : 6,		CONFIG : 'N U T, 0, 0, 0',
	X =  -100.833  mm,	Y =   -368.014  mm,	Z =   -242.162  mm,
	W =  90.000 deg,	P =   0.000 deg,	R =   90.000 deg
};
P[1900]{
   GP1:
	UF : 0, UT : 6,		CONFIG : 'N U T, 0, 0, 0',
	X =  -101.773  mm,	Y =   -368.546  mm,	Z =   -242.137  mm,
	W =  90.000 deg,	P =   0.000 deg,	R =   90.000 deg
};
P[1901]{
   GP1:
	UF : 0, UT : 6,		CONFIG : 'N U T, 0, 0, 0',
	X =  -103.649  mm,	Y =   -369.684  mm,	Z =   -242.269  mm,
	W =  90.000 deg,	P =   0.000 deg,	R =   90.000 deg
};
P[1902]{
   GP1:
	UF : 0, UT : 6,		CONFIG : 'N U T, 0, 0, 0',
	X =  -106.020  mm,	Y =   -370.935  mm,	Z =   -241.983  mm,
	W =  90.000 deg,	P =   0.000 deg,	R =   90.000 deg
};
P[1903]{
   GP1:
	UF : 0, UT : 6,		CONFIG : 'N U T, 0, 0, 0',
	X =  -106.783  mm,	Y =   -371.407  mm,	Z =   -242.060  mm,
	W =  90.000 deg,	P =   0.000 deg,	R =   90.000 deg
};
P[1904]{
   GP1:
	UF : 0, UT : 6,		CONFIG : 'N U T, 0, 0, 0',
	X =  -108.729  mm,	Y =   -372.660  mm,	Z =   -242.373  mm,
	W =  90.000 deg,	P =   0.000 deg,	R =   90.000 deg
};
P[1905]{
   GP1:
	UF : 0, UT : 6,		CONFIG : 'N U T, 0, 0, 0',
	X =  -109.547  mm,	Y =   -373.119  mm,	Z =   -242.341  mm,
	W =  90.000 deg,	P =   0.000 deg,	R =   90.000 deg
};
P[1906]{
   GP1:
	UF : 0, UT : 6,		CONFIG : 'N U T, 0, 0, 0',
	X =  -110.237  mm,	Y =   -373.518  mm,	Z =   -242.343  mm,
	W =  90.000 deg,	P =   0.000 deg,	R =   90.000 deg
};
P[1907]{
   GP1:
	UF : 0, UT : 6,		CONFIG : 'N U T, 0, 0, 0',
	X =  -114.668  mm,	Y =   -376.086  mm,	Z =   -242.364  mm,
	W =  90.000 deg,	P =   0.000 deg,	R =   90.000 deg
};
P[1908]{
   GP1:
	UF : 0, UT : 6,		CONFIG : 'N U T, 0, 0, 0',
	X =  -116.212  mm,	Y =   -376.798  mm,	Z =   -241.932  mm,
	W =  90.000 deg,	P =   0.000 deg,	R =   90.000 deg
};
P[1909]{
   GP1:
	UF : 0, UT : 6,		CONFIG : 'N U T, 0, 0, 0',
	X =  -117.073  mm,	Y =   -377.316  mm,	Z =   -241.982  mm,
	W =  90.000 deg,	P =   0.000 deg,	R =   90.000 deg
};
P[1910]{
   GP1:
	UF : 0, UT : 6,		CONFIG : 'N U T, 0, 0, 0',
	X =  -118.913  mm,	Y =   -378.468  mm,	Z =   -242.196  mm,
	W =  90.000 deg,	P =   0.000 deg,	R =   90.000 deg
};
P[1911]{
   GP1:
	UF : 0, UT : 6,		CONFIG : 'N U T, 0, 0, 0',
	X =  -121.499  mm,	Y =   -379.895  mm,	Z =   -242.038  mm,
	W =  90.000 deg,	P =   0.000 deg,	R =   90.000 deg
};
P[1912]{
   GP1:
	UF : 0, UT : 6,		CONFIG : 'N U T, 0, 0, 0',
	X =  -122.885  mm,	Y =   -380.831  mm,	Z =   -242.368  mm,
	W =  90.000 deg,	P =   0.000 deg,	R =   90.000 deg
};
P[1913]{
   GP1:
	UF : 0, UT : 6,		CONFIG : 'N U T, 0, 0, 0',
	X =  -124.769  mm,	Y =   -381.844  mm,	Z =   -242.186  mm,
	W =  90.000 deg,	P =   0.000 deg,	R =   90.000 deg
};
P[1914]{
   GP1:
	UF : 0, UT : 6,		CONFIG : 'N U T, 0, 0, 0',
	X =  -125.945  mm,	Y =   -382.551  mm,	Z =   -242.253  mm,
	W =  90.000 deg,	P =   0.000 deg,	R =   90.000 deg
};
P[1915]{
   GP1:
	UF : 0, UT : 6,		CONFIG : 'N U T, 0, 0, 0',
	X =  -127.551  mm,	Y =   -383.390  mm,	Z =   -242.039  mm,
	W =  90.000 deg,	P =   0.000 deg,	R =   90.000 deg
};
P[1916]{
   GP1:
	UF : 0, UT : 6,		CONFIG : 'N U T, 0, 0, 0',
	X =  -130.132  mm,	Y =   -385.023  mm,	Z =   -242.185  mm,
	W =  90.000 deg,	P =   0.000 deg,	R =   90.000 deg
};
P[1917]{
   GP1:
	UF : 0, UT : 6,		CONFIG : 'N U T, 0, 0, 0',
	X =  -131.227  mm,	Y =   -385.866  mm,	Z =   -242.303  mm,
	W =  90.000 deg,	P =   0.000 deg,	R =   90.000 deg
};
P[1918]{
   GP1:
	UF : 0, UT : 6,		CONFIG : 'N U T, 0, 0, 0',
	X =  -132.088  mm,	Y =   -386.525  mm,	Z =   -242.239  mm,
	W =  90.000 deg,	P =   0.000 deg,	R =   90.000 deg
};
P[1919]{
   GP1:
	UF : 0, UT : 6,		CONFIG : 'N U T, 0, 0, 0',
	X =  -133.466  mm,	Y =   -388.038  mm,	Z =   -242.271  mm,
	W =  90.000 deg,	P =   0.000 deg,	R =   90.000 deg
};
P[1920]{
   GP1:
	UF : 0, UT : 6,		CONFIG : 'N U T, 0, 0, 0',
	X =  -134.348  mm,	Y =   -388.919  mm,	Z =   -241.887  mm,
	W =  90.000 deg,	P =   0.000 deg,	R =   90.000 deg
};
P[1921]{
   GP1:
	UF : 0, UT : 6,		CONFIG : 'N U T, 0, 0, 0',
	X =  -135.411  mm,	Y =   -391.196  mm,	Z =   -242.232  mm,
	W =  90.000 deg,	P =   0.000 deg,	R =   90.000 deg
};
P[1922]{
   GP1:
	UF : 0, UT : 6,		CONFIG : 'N U T, 0, 0, 0',
	X =  -136.326  mm,	Y =   -394.925  mm,	Z =   -242.365  mm,
	W =  90.000 deg,	P =   0.000 deg,	R =   90.000 deg
};
P[1923]{
   GP1:
	UF : 0, UT : 6,		CONFIG : 'N U T, 0, 0, 0',
	X =  -136.247  mm,	Y =   -398.620  mm,	Z =   -242.249  mm,
	W =  90.000 deg,	P =   0.000 deg,	R =   90.000 deg
};
P[1924]{
   GP1:
	UF : 0, UT : 6,		CONFIG : 'N U T, 0, 0, 0',
	X =  -135.816  mm,	Y =   -400.863  mm,	Z =   -242.002  mm,
	W =  90.000 deg,	P =   0.000 deg,	R =   90.000 deg
};
P[1925]{
   GP1:
	UF : 0, UT : 6,		CONFIG : 'N U T, 0, 0, 0',
	X =  -135.266  mm,	Y =   -401.987  mm,	Z =   -242.122  mm,
	W =  90.000 deg,	P =   0.000 deg,	R =   90.000 deg
};
P[1926]{
   GP1:
	UF : 0, UT : 6,		CONFIG : 'N U T, 0, 0, 0',
	X =  -134.300  mm,	Y =   -404.089  mm,	Z =   -241.942  mm,
	W =  90.000 deg,	P =   0.000 deg,	R =   90.000 deg
};
P[1927]{
   GP1:
	UF : 0, UT : 6,		CONFIG : 'N U T, 0, 0, 0',
	X =  -133.482  mm,	Y =   -405.279  mm,	Z =   -242.261  mm,
	W =  90.000 deg,	P =   0.000 deg,	R =   90.000 deg
};
P[1928]{
   GP1:
	UF : 0, UT : 6,		CONFIG : 'N U T, 0, 0, 0',
	X =  -131.694  mm,	Y =   -408.330  mm,	Z =   -242.324  mm,
	W =  90.000 deg,	P =   0.000 deg,	R =   90.000 deg
};
P[1929]{
   GP1:
	UF : 0, UT : 6,		CONFIG : 'N U T, 0, 0, 0',
	X =  -130.079  mm,	Y =   -411.086  mm,	Z =   -242.381  mm,
	W =  90.000 deg,	P =   0.000 deg,	R =   90.000 deg
};
P[1930]{
   GP1:
	UF : 0, UT : 6,		CONFIG : 'N U T, 0, 0, 0',
	X =  -128.240  mm,	Y =   -414.310  mm,	Z =   -242.326  mm,
	W =  90.000 deg,	P =   0.000 deg,	R =   90.000 deg
};
P[1931]{
   GP1:
	UF : 0, UT : 6,		CONFIG : 'N U T, 0, 0, 0',
	X =  -127.549  mm,	Y =   -415.646  mm,	Z =   -242.131  mm,
	W =  90.000 deg,	P =   0.000 deg,	R =   90.000 deg
};
P[1932]{
   GP1:
	UF : 0, UT : 6,		CONFIG : 'N U T, 0, 0, 0',
	X =  -125.189  mm,	Y =   -419.819  mm,	Z =   -242.012  mm,
	W =  90.000 deg,	P =   0.000 deg,	R =   90.000 deg
};
P[1933]{
   GP1:
	UF : 0, UT : 6,		CONFIG : 'N U T, 0, 0, 0',
	X =  -124.577  mm,	Y =   -420.708  mm,	Z =   -242.252  mm,
	W =  90.000 deg,	P =   0.000 deg,	R =   90.000 deg
};
P[1934]{
   GP1:
	UF : 0, UT : 6,		CONFIG : 'N U T, 0, 0, 0',
	X =  -123.832  mm,	Y =   -421.983  mm,	Z =   -242.272  mm,
	W =  90.000 deg,	P =   0.000 deg,	R =   90.000 deg
};
P[1935]{
   GP1:
	UF : 0, UT : 6,		CONFIG : 'N U T, 0, 0, 0',
	X =  -123.457  mm,	Y =   -422.727  mm,	Z =   -242.140  mm,
	W =  90.000 deg,	P =   0.000 deg,	R =   90.000 deg
};
P[1936]{
   GP1:
	UF : 0, UT : 6,		CONFIG : 'N U T, 0, 0, 0',
	X =  -123.050  mm,	Y =   -423.372  mm,	Z =   -242.224  mm,
	W =  90.000 deg,	P =   0.000 deg,	R =   90.000 deg
};
P[1937]{
   GP1:
	UF : 0, UT : 6,		CONFIG : 'N U T, 0, 0, 0',
	X =  -121.937  mm,	Y =   -425.271  mm,	Z =   -242.262  mm,
	W =  90.000 deg,	P =   0.000 deg,	R =   90.000 deg
};
P[1938]{
   GP1:
	UF : 0, UT : 6,		CONFIG : 'N U T, 0, 0, 0',
	X =  -119.854  mm,	Y =   -428.799  mm,	Z =   -242.377  mm,
	W =  90.000 deg,	P =   0.000 deg,	R =   90.000 deg
};
P[1939]{
   GP1:
	UF : 0, UT : 6,		CONFIG : 'N U T, 0, 0, 0',
	X =  -118.300  mm,	Y =   -431.529  mm,	Z =   -242.320  mm,
	W =  90.000 deg,	P =   0.000 deg,	R =   90.000 deg
};
P[1940]{
   GP1:
	UF : 0, UT : 6,		CONFIG : 'N U T, 0, 0, 0',
	X =  -118.043  mm,	Y =   -432.194  mm,	Z =   -242.014  mm,
	W =  90.000 deg,	P =   0.000 deg,	R =   90.000 deg
};
P[1941]{
   GP1:
	UF : 0, UT : 6,		CONFIG : 'N U T, 0, 0, 0',
	X =  -117.513  mm,	Y =   -433.045  mm,	Z =   -242.107  mm,
	W =  90.000 deg,	P =   0.000 deg,	R =   90.000 deg
};
P[1942]{
   GP1:
	UF : 0, UT : 6,		CONFIG : 'N U T, 0, 0, 0',
	X =  -116.847  mm,	Y =   -434.179  mm,	Z =   -242.135  mm,
	W =  90.000 deg,	P =   0.000 deg,	R =   90.000 deg
};
P[1943]{
   GP1:
	UF : 0, UT : 6,		CONFIG : 'N U T, 0, 0, 0',
	X =  -115.505  mm,	Y =   -436.472  mm,	Z =   -242.178  mm,
	W =  90.000 deg,	P =   0.000 deg,	R =   90.000 deg
};
P[1944]{
   GP1:
	UF : 0, UT : 6,		CONFIG : 'N U T, 0, 0, 0',
	X =  -114.446  mm,	Y =   -438.381  mm,	Z =   -242.071  mm,
	W =  90.000 deg,	P =   0.000 deg,	R =   90.000 deg
};
P[1945]{
   GP1:
	UF : 0, UT : 6,		CONFIG : 'N U T, 0, 0, 0',
	X =  -113.710  mm,	Y =   -439.575  mm,	Z =   -242.187  mm,
	W =  90.000 deg,	P =   0.000 deg,	R =   90.000 deg
};
P[1946]{
   GP1:
	UF : 0, UT : 6,		CONFIG : 'N U T, 0, 0, 0',
	X =  -113.046  mm,	Y =   -440.704  mm,	Z =   -242.213  mm,
	W =  90.000 deg,	P =   0.000 deg,	R =   90.000 deg
};
P[1947]{
   GP1:
	UF : 0, UT : 6,		CONFIG : 'N U T, 0, 0, 0',
	X =  -112.208  mm,	Y =   -442.253  mm,	Z =   -242.080  mm,
	W =  90.000 deg,	P =   0.000 deg,	R =   90.000 deg
};
P[1948]{
   GP1:
	UF : 0, UT : 6,		CONFIG : 'N U T, 0, 0, 0',
	X =  -108.792  mm,	Y =   -448.162  mm,	Z =   -242.089  mm,
	W =  90.000 deg,	P =   0.000 deg,	R =   90.000 deg
};
P[1949]{
   GP1:
	UF : 0, UT : 6,		CONFIG : 'N U T, 0, 0, 0',
	X =  -107.043  mm,	Y =   -450.985  mm,	Z =   -242.378  mm,
	W =  90.000 deg,	P =   0.000 deg,	R =   90.000 deg
};
P[1950]{
   GP1:
	UF : 0, UT : 6,		CONFIG : 'N U T, 0, 0, 0',
	X =  -105.691  mm,	Y =   -453.415  mm,	Z =   -242.254  mm,
	W =  90.000 deg,	P =   0.000 deg,	R =   90.000 deg
};
P[1951]{
   GP1:
	UF : 0, UT : 6,		CONFIG : 'N U T, 0, 0, 0',
	X =  -104.183  mm,	Y =   -455.979  mm,	Z =   -242.321  mm,
	W =  90.000 deg,	P =   0.000 deg,	R =   90.000 deg
};
P[1952]{
   GP1:
	UF : 0, UT : 6,		CONFIG : 'N U T, 0, 0, 0',
	X =  -102.431  mm,	Y =   -459.271  mm,	Z =   -241.960  mm,
	W =  90.000 deg,	P =   0.000 deg,	R =   90.000 deg
};
P[1953]{
   GP1:
	UF : 0, UT : 6,		CONFIG : 'N U T, 0, 0, 0',
	X =  -100.015  mm,	Y =   -463.183  mm,	Z =   -242.340  mm,
	W =  90.000 deg,	P =   0.000 deg,	R =   90.000 deg
};
P[1954]{
   GP1:
	UF : 0, UT : 6,		CONFIG : 'N U T, 0, 0, 0',
	X =  -98.421  mm,	Y =   -465.947  mm,	Z =   -242.336  mm,
	W =  90.000 deg,	P =   0.000 deg,	R =   90.000 deg
};
P[1955]{
   GP1:
	UF : 0, UT : 6,		CONFIG : 'N U T, 0, 0, 0',
	X =  -97.380  mm,	Y =   -467.760  mm,	Z =   -242.321  mm,
	W =  90.000 deg,	P =   0.000 deg,	R =   90.000 deg
};
P[1956]{
   GP1:
	UF : 0, UT : 6,		CONFIG : 'N U T, 0, 0, 0',
	X =  -96.175  mm,	Y =   -470.032  mm,	Z =   -242.063  mm,
	W =  90.000 deg,	P =   0.000 deg,	R =   90.000 deg
};
P[1957]{
   GP1:
	UF : 0, UT : 6,		CONFIG : 'N U T, 0, 0, 0',
	X =  -94.979  mm,	Y =   -471.893  mm,	Z =   -242.357  mm,
	W =  90.000 deg,	P =   0.000 deg,	R =   90.000 deg
};
P[1958]{
   GP1:
	UF : 0, UT : 6,		CONFIG : 'N U T, 0, 0, 0',
	X =  -92.649  mm,	Y =   -475.994  mm,	Z =   -242.267  mm,
	W =  90.000 deg,	P =   0.000 deg,	R =   90.000 deg
};
P[1959]{
   GP1:
	UF : 0, UT : 6,		CONFIG : 'N U T, 0, 0, 0',
	X =  -91.948  mm,	Y =   -477.135  mm,	Z =   -242.366  mm,
	W =  90.000 deg,	P =   0.000 deg,	R =   90.000 deg
};
P[1960]{
   GP1:
	UF : 0, UT : 6,		CONFIG : 'N U T, 0, 0, 0',
	X =  -91.530  mm,	Y =   -478.071  mm,	Z =   -242.070  mm,
	W =  90.000 deg,	P =   0.000 deg,	R =   90.000 deg
};
P[1961]{
   GP1:
	UF : 0, UT : 6,		CONFIG : 'N U T, 0, 0, 0',
	X =  -90.644  mm,	Y =   -479.703  mm,	Z =   -241.933  mm,
	W =  90.000 deg,	P =   0.000 deg,	R =   90.000 deg
};
P[1962]{
   GP1:
	UF : 0, UT : 6,		CONFIG : 'N U T, 0, 0, 0',
	X =  -89.633  mm,	Y =   -481.183  mm,	Z =   -242.314  mm,
	W =  90.000 deg,	P =   0.000 deg,	R =   90.000 deg
};
P[1963]{
   GP1:
	UF : 0, UT : 6,		CONFIG : 'N U T, 0, 0, 0',
	X =  -89.254  mm,	Y =   -481.875  mm,	Z =   -242.265  mm,
	W =  90.000 deg,	P =   0.000 deg,	R =   90.000 deg
};
P[1964]{
   GP1:
	UF : 0, UT : 6,		CONFIG : 'N U T, 0, 0, 0',
	X =  -88.286  mm,	Y =   -483.574  mm,	Z =   -242.233  mm,
	W =  90.000 deg,	P =   0.000 deg,	R =   90.000 deg
};
P[1965]{
   GP1:
	UF : 0, UT : 6,		CONFIG : 'N U T, 0, 0, 0',
	X =  -87.458  mm,	Y =   -485.013  mm,	Z =   -242.226  mm,
	W =  90.000 deg,	P =   0.000 deg,	R =   90.000 deg
};
P[1966]{
   GP1:
	UF : 0, UT : 6,		CONFIG : 'N U T, 0, 0, 0',
	X =  -84.387  mm,	Y =   -490.325  mm,	Z =   -242.235  mm,
	W =  90.000 deg,	P =   0.000 deg,	R =   90.000 deg
};
P[1967]{
   GP1:
	UF : 0, UT : 6,		CONFIG : 'N U T, 0, 0, 0',
	X =  -83.903  mm,	Y =   -491.409  mm,	Z =   -241.890  mm,
	W =  90.000 deg,	P =   0.000 deg,	R =   90.000 deg
};
P[1968]{
   GP1:
	UF : 0, UT : 6,		CONFIG : 'N U T, 0, 0, 0',
	X =  -83.327  mm,	Y =   -492.157  mm,	Z =   -242.242  mm,
	W =  90.000 deg,	P =   0.000 deg,	R =   90.000 deg
};
P[1969]{
   GP1:
	UF : 0, UT : 6,		CONFIG : 'N U T, 0, 0, 0',
	X =  -82.317  mm,	Y =   -493.895  mm,	Z =   -242.258  mm,
	W =  90.000 deg,	P =   0.000 deg,	R =   90.000 deg
};
P[1970]{
   GP1:
	UF : 0, UT : 6,		CONFIG : 'N U T, 0, 0, 0',
	X =  -81.466  mm,	Y =   -495.493  mm,	Z =   -242.083  mm,
	W =  90.000 deg,	P =   0.000 deg,	R =   90.000 deg
};
P[1971]{
   GP1:
	UF : 0, UT : 6,		CONFIG : 'N U T, 0, 0, 0',
	X =  -80.816  mm,	Y =   -496.558  mm,	Z =   -242.166  mm,
	W =  90.000 deg,	P =   0.000 deg,	R =   90.000 deg
};
P[1972]{
   GP1:
	UF : 0, UT : 6,		CONFIG : 'N U T, 0, 0, 0',
	X =  -80.431  mm,	Y =   -497.119  mm,	Z =   -242.316  mm,
	W =  90.000 deg,	P =   0.000 deg,	R =   90.000 deg
};
P[1973]{
   GP1:
	UF : 0, UT : 6,		CONFIG : 'N U T, 0, 0, 0',
	X =  -78.677  mm,	Y =   -500.249  mm,	Z =   -242.187  mm,
	W =  90.000 deg,	P =   0.000 deg,	R =   90.000 deg
};
P[1974]{
   GP1:
	UF : 0, UT : 6,		CONFIG : 'N U T, 0, 0, 0',
	X =  -77.883  mm,	Y =   -501.594  mm,	Z =   -242.229  mm,
	W =  90.000 deg,	P =   0.000 deg,	R =   90.000 deg
};
P[1975]{
   GP1:
	UF : 0, UT : 6,		CONFIG : 'N U T, 0, 0, 0',
	X =  -77.409  mm,	Y =   -502.426  mm,	Z =   -242.215  mm,
	W =  90.000 deg,	P =   0.000 deg,	R =   90.000 deg
};
P[1976]{
   GP1:
	UF : 0, UT : 6,		CONFIG : 'N U T, 0, 0, 0',
	X =  -76.863  mm,	Y =   -503.370  mm,	Z =   -242.217  mm,
	W =  90.000 deg,	P =   0.000 deg,	R =   90.000 deg
};
P[1977]{
   GP1:
	UF : 0, UT : 6,		CONFIG : 'N U T, 0, 0, 0',
	X =  -76.103  mm,	Y =   -504.693  mm,	Z =   -242.207  mm,
	W =  90.000 deg,	P =   0.000 deg,	R =   90.000 deg
};
P[1978]{
   GP1:
	UF : 0, UT : 6,		CONFIG : 'N U T, 0, 0, 0',
	X =  -74.627  mm,	Y =   -507.170  mm,	Z =   -242.317  mm,
	W =  90.000 deg,	P =   0.000 deg,	R =   90.000 deg
};
P[1979]{
   GP1:
	UF : 0, UT : 6,		CONFIG : 'N U T, 0, 0, 0',
	X =  -73.285  mm,	Y =   -509.802  mm,	Z =   -241.887  mm,
	W =  90.000 deg,	P =   0.000 deg,	R =   90.000 deg
};
P[1980]{
   GP1:
	UF : 0, UT : 6,		CONFIG : 'N U T, 0, 0, 0',
	X =  -72.685  mm,	Y =   -510.745  mm,	Z =   -242.022  mm,
	W =  90.000 deg,	P =   0.000 deg,	R =   90.000 deg
};
P[1981]{
   GP1:
	UF : 0, UT : 6,		CONFIG : 'N U T, 0, 0, 0',
	X =  -71.787  mm,	Y =   -512.090  mm,	Z =   -242.315  mm,
	W =  90.000 deg,	P =   0.000 deg,	R =   90.000 deg
};
P[1982]{
   GP1:
	UF : 0, UT : 6,		CONFIG : 'N U T, 0, 0, 0',
	X =  -71.170  mm,	Y =   -513.458  mm,	Z =   -241.896  mm,
	W =  90.000 deg,	P =   0.000 deg,	R =   90.000 deg
};
P[1983]{
   GP1:
	UF : 0, UT : 6,		CONFIG : 'N U T, 0, 0, 0',
	X =  -70.124  mm,	Y =   -515.227  mm,	Z =   -241.956  mm,
	W =  90.000 deg,	P =   0.000 deg,	R =   90.000 deg
};
P[1984]{
   GP1:
	UF : 0, UT : 6,		CONFIG : 'N U T, 0, 0, 0',
	X =  -69.550  mm,	Y =   -515.988  mm,	Z =   -242.282  mm,
	W =  90.000 deg,	P =   0.000 deg,	R =   90.000 deg
};
P[1985]{
   GP1:
	UF : 0, UT : 6,		CONFIG : 'N U T, 0, 0, 0',
	X =  -66.961  mm,	Y =   -520.444  mm,	Z =   -242.322  mm,
	W =  90.000 deg,	P =   0.000 deg,	R =   90.000 deg
};
P[1986]{
   GP1:
	UF : 0, UT : 6,		CONFIG : 'N U T, 0, 0, 0',
	X =  -66.672  mm,	Y =   -521.053  mm,	Z =   -242.171  mm,
	W =  90.000 deg,	P =   0.000 deg,	R =   90.000 deg
};
P[1987]{
   GP1:
	UF : 0, UT : 6,		CONFIG : 'N U T, 0, 0, 0',
	X =  -66.153  mm,	Y =   -522.027  mm,	Z =   -242.065  mm,
	W =  90.000 deg,	P =   0.000 deg,	R =   90.000 deg
};
P[1988]{
   GP1:
	UF : 0, UT : 6,		CONFIG : 'N U T, 0, 0, 0',
	X =  -65.653  mm,	Y =   -522.855  mm,	Z =   -242.118  mm,
	W =  90.000 deg,	P =   0.000 deg,	R =   90.000 deg
};
P[1989]{
   GP1:
	UF : 0, UT : 6,		CONFIG : 'N U T, 0, 0, 0',
	X =  -64.107  mm,	Y =   -525.415  mm,	Z =   -242.284  mm,
	W =  90.000 deg,	P =   0.000 deg,	R =   90.000 deg
};
P[1990]{
   GP1:
	UF : 0, UT : 6,		CONFIG : 'N U T, 0, 0, 0',
	X =  -63.122  mm,	Y =   -527.064  mm,	Z =   -242.361  mm,
	W =  90.000 deg,	P =   0.000 deg,	R =   90.000 deg
};
P[1991]{
   GP1:
	UF : 0, UT : 6,		CONFIG : 'N U T, 0, 0, 0',
	X =  -62.195  mm,	Y =   -528.909  mm,	Z =   -242.026  mm,
	W =  90.000 deg,	P =   0.000 deg,	R =   90.000 deg
};
P[1992]{
   GP1:
	UF : 0, UT : 6,		CONFIG : 'N U T, 0, 0, 0',
	X =  -61.241  mm,	Y =   -530.341  mm,	Z =   -242.337  mm,
	W =  90.000 deg,	P =   0.000 deg,	R =   90.000 deg
};
P[1993]{
   GP1:
	UF : 0, UT : 6,		CONFIG : 'N U T, 0, 0, 0',
	X =  -60.753  mm,	Y =   -531.181  mm,	Z =   -242.343  mm,
	W =  90.000 deg,	P =   0.000 deg,	R =   90.000 deg
};
P[1994]{
   GP1:
	UF : 0, UT : 6,		CONFIG : 'N U T, 0, 0, 0',
	X =  -59.427  mm,	Y =   -533.487  mm,	Z =   -242.329  mm,
	W =  90.000 deg,	P =   0.000 deg,	R =   90.000 deg
};
P[1995]{
   GP1:
	UF : 0, UT : 6,		CONFIG : 'N U T, 0, 0, 0',
	X =  -59.089  mm,	Y =   -534.262  mm,	Z =   -242.065  mm,
	W =  90.000 deg,	P =   0.000 deg,	R =   90.000 deg
};
P[1996]{
   GP1:
	UF : 0, UT : 6,		CONFIG : 'N U T, 0, 0, 0',
	X =  -58.195  mm,	Y =   -535.680  mm,	Z =   -242.248  mm,
	W =  90.000 deg,	P =   0.000 deg,	R =   90.000 deg
};
P[1997]{
   GP1:
	UF : 0, UT : 6,		CONFIG : 'N U T, 0, 0, 0',
	X =  -57.057  mm,	Y =   -537.887  mm,	Z =   -241.916  mm,
	W =  90.000 deg,	P =   0.000 deg,	R =   90.000 deg
};
P[1998]{
   GP1:
	UF : 0, UT : 6,		CONFIG : 'N U T, 0, 0, 0',
	X =  -56.036  mm,	Y =   -539.493  mm,	Z =   -242.143  mm,
	W =  90.000 deg,	P =   0.000 deg,	R =   90.000 deg
};
P[1999]{
   GP1:
	UF : 0, UT : 6,		CONFIG : 'N U T, 0, 0, 0',
	X =  -55.650  mm,	Y =   -540.063  mm,	Z =   -242.282  mm,
	W =  90.000 deg,	P =   0.000 deg,	R =   90.000 deg
};
P[2000]{
   GP1:
	UF : 0, UT : 6,		CONFIG : 'N U T, 0, 0, 0',
	X =  -54.758  mm,	Y =   -541.837  mm,	Z =   -241.959  mm,
	W =  90.000 deg,	P =   0.000 deg,	R =   90.000 deg
};
P[2001]{
   GP1:
	UF : 0, UT : 6,		CONFIG : 'N U T, 0, 0, 0',
	X =  -53.797  mm,	Y =   -543.504  mm,	Z =   -241.955  mm,
	W =  90.000 deg,	P =   0.000 deg,	R =   90.000 deg
};
P[2002]{
   GP1:
	UF : 0, UT : 6,		CONFIG : 'N U T, 0, 0, 0',
	X =  -52.082  mm,	Y =   -546.340  mm,	Z =   -242.144  mm,
	W =  90.000 deg,	P =   0.000 deg,	R =   90.000 deg
};
P[2003]{
   GP1:
	UF : 0, UT : 6,		CONFIG : 'N U T, 0, 0, 0',
	X =  -49.997  mm,	Y =   -550.038  mm,	Z =   -242.021  mm,
	W =  90.000 deg,	P =   0.000 deg,	R =   90.000 deg
};
P[2004]{
   GP1:
	UF : 0, UT : 6,		CONFIG : 'N U T, 0, 0, 0',
	X =  -49.606  mm,	Y =   -550.468  mm,	Z =   -242.371  mm,
	W =  90.000 deg,	P =   0.000 deg,	R =   90.000 deg
};
P[2005]{
   GP1:
	UF : 0, UT : 6,		CONFIG : 'N U T, 0, 0, 0',
	X =  -44.260  mm,	Y =   -559.844  mm,	Z =   -242.206  mm,
	W =  90.000 deg,	P =   0.000 deg,	R =   90.000 deg
};
P[2006]{
   GP1:
	UF : 0, UT : 6,		CONFIG : 'N U T, 0, 0, 0',
	X =  -43.583  mm,	Y =   -561.141  mm,	Z =   -242.029  mm,
	W =  90.000 deg,	P =   0.000 deg,	R =   90.000 deg
};
P[2007]{
   GP1:
	UF : 0, UT : 6,		CONFIG : 'N U T, 0, 0, 0',
	X =  -42.612  mm,	Y =   -562.856  mm,	Z =   -241.985  mm,
	W =  90.000 deg,	P =   0.000 deg,	R =   90.000 deg
};
P[2008]{
   GP1:
	UF : 0, UT : 6,		CONFIG : 'N U T, 0, 0, 0',
	X =  -41.121  mm,	Y =   -565.420  mm,	Z =   -242.009  mm,
	W =  90.000 deg,	P =   0.000 deg,	R =   90.000 deg
};
P[2009]{
   GP1:
	UF : 0, UT : 6,		CONFIG : 'N U T, 0, 0, 0',
	X =  -39.774  mm,	Y =   -567.562  mm,	Z =   -242.277  mm,
	W =  90.000 deg,	P =   0.000 deg,	R =   90.000 deg
};
P[2010]{
   GP1:
	UF : 0, UT : 6,		CONFIG : 'N U T, 0, 0, 0',
	X =  -38.757  mm,	Y =   -569.352  mm,	Z =   -242.236  mm,
	W =  90.000 deg,	P =   0.000 deg,	R =   90.000 deg
};
P[2011]{
   GP1:
	UF : 0, UT : 6,		CONFIG : 'N U T, 0, 0, 0',
	X =  -38.229  mm,	Y =   -570.446  mm,	Z =   -241.985  mm,
	W =  90.000 deg,	P =   0.000 deg,	R =   90.000 deg
};
P[2012]{
   GP1:
	UF : 0, UT : 6,		CONFIG : 'N U T, 0, 0, 0',
	X =  -37.769  mm,	Y =   -571.224  mm,	Z =   -242.011  mm,
	W =  90.000 deg,	P =   0.000 deg,	R =   90.000 deg
};
P[2013]{
   GP1:
	UF : 0, UT : 6,		CONFIG : 'N U T, 0, 0, 0',
	X =  -36.718  mm,	Y =   -572.837  mm,	Z =   -242.301  mm,
	W =  90.000 deg,	P =   0.000 deg,	R =   90.000 deg
};
P[2014]{
   GP1:
	UF : 0, UT : 6,		CONFIG : 'N U T, 0, 0, 0',
	X =  -35.995  mm,	Y =   -574.221  mm,	Z =   -242.119  mm,
	W =  90.000 deg,	P =   0.000 deg,	R =   90.000 deg
};
P[2015]{
   GP1:
	UF : 0, UT : 6,		CONFIG : 'N U T, 0, 0, 0',
	X =  -34.219  mm,	Y =   -577.297  mm,	Z =   -242.116  mm,
	W =  90.000 deg,	P =   0.000 deg,	R =   90.000 deg
};
P[2016]{
   GP1:
	UF : 0, UT : 6,		CONFIG : 'N U T, 0, 0, 0',
	X =  -32.556  mm,	Y =   -580.109  mm,	Z =   -242.211  mm,
	W =  90.000 deg,	P =   0.000 deg,	R =   90.000 deg
};
P[2017]{
   GP1:
	UF : 0, UT : 6,		CONFIG : 'N U T, 0, 0, 0',
	X =  -31.904  mm,	Y =   -581.149  mm,	Z =   -242.338  mm,
	W =  90.000 deg,	P =   0.000 deg,	R =   90.000 deg
};
P[2018]{
   GP1:
	UF : 0, UT : 6,		CONFIG : 'N U T, 0, 0, 0',
	X =  -29.965  mm,	Y =   -584.518  mm,	Z =   -242.322  mm,
	W =  90.000 deg,	P =   0.000 deg,	R =   90.000 deg
};
P[2019]{
   GP1:
	UF : 0, UT : 6,		CONFIG : 'N U T, 0, 0, 0',
	X =  -27.084  mm,	Y =   -589.492  mm,	Z =   -242.342  mm,
	W =  90.000 deg,	P =   0.000 deg,	R =   90.000 deg
};
P[2020]{
   GP1:
	UF : 0, UT : 6,		CONFIG : 'N U T, 0, 0, 0',
	X =  -24.081  mm,	Y =   -594.752  mm,	Z =   -242.260  mm,
	W =  90.000 deg,	P =   0.000 deg,	R =   90.000 deg
};
P[2021]{
   GP1:
	UF : 0, UT : 6,		CONFIG : 'N U T, 0, 0, 0',
	X =  -22.944  mm,	Y =   -596.761  mm,	Z =   -242.205  mm,
	W =  90.000 deg,	P =   0.000 deg,	R =   90.000 deg
};
P[2022]{
   GP1:
	UF : 0, UT : 6,		CONFIG : 'N U T, 0, 0, 0',
	X =  -20.707  mm,	Y =   -600.657  mm,	Z =   -242.176  mm,
	W =  90.000 deg,	P =   0.000 deg,	R =   90.000 deg
};
P[2023]{
   GP1:
	UF : 0, UT : 6,		CONFIG : 'N U T, 0, 0, 0',
	X =  -19.674  mm,	Y =   -602.315  mm,	Z =   -242.358  mm,
	W =  90.000 deg,	P =   0.000 deg,	R =   90.000 deg
};
P[2024]{
   GP1:
	UF : 0, UT : 6,		CONFIG : 'N U T, 0, 0, 0',
	X =  -19.432  mm,	Y =   -602.949  mm,	Z =   -242.058  mm,
	W =  90.000 deg,	P =   0.000 deg,	R =   90.000 deg
};
P[2025]{
   GP1:
	UF : 0, UT : 6,		CONFIG : 'N U T, 0, 0, 0',
	X =  -18.757  mm,	Y =   -603.924  mm,	Z =   -242.329  mm,
	W =  90.000 deg,	P =   0.000 deg,	R =   90.000 deg
};
P[2026]{
   GP1:
	UF : 0, UT : 6,		CONFIG : 'N U T, 0, 0, 0',
	X =  -17.811  mm,	Y =   -605.645  mm,	Z =   -242.216  mm,
	W =  90.000 deg,	P =   0.000 deg,	R =   90.000 deg
};
P[2027]{
   GP1:
	UF : 0, UT : 6,		CONFIG : 'N U T, 0, 0, 0',
	X =  -17.203  mm,	Y =   -606.831  mm,	Z =   -242.028  mm,
	W =  90.000 deg,	P =   0.000 deg,	R =   90.000 deg
};
P[2028]{
   GP1:
	UF : 0, UT : 6,		CONFIG : 'N U T, 0, 0, 0',
	X =  -15.610  mm,	Y =   -609.372  mm,	Z =   -242.334  mm,
	W =  90.000 deg,	P =   0.000 deg,	R =   90.000 deg
};
P[2029]{
   GP1:
	UF : 0, UT : 6,		CONFIG : 'N U T, 0, 0, 0',
	X =  -15.365  mm,	Y =   -610.026  mm,	Z =   -242.011  mm,
	W =  90.000 deg,	P =   0.000 deg,	R =   90.000 deg
};
P[2030]{
   GP1:
	UF : 0, UT : 6,		CONFIG : 'N U T, 0, 0, 0',
	X =  -13.950  mm,	Y =   -612.403  mm,	Z =   -242.116  mm,
	W =  90.000 deg,	P =   0.000 deg,	R =   90.000 deg
};
P[2031]{
   GP1:
	UF : 0, UT : 6,		CONFIG : 'N U T, 0, 0, 0',
	X =  -13.438  mm,	Y =   -613.124  mm,	Z =   -242.349  mm,
	W =  90.000 deg,	P =   0.000 deg,	R =   90.000 deg
};
P[2032]{
   GP1:
	UF : 0, UT : 6,		CONFIG : 'N U T, 0, 0, 0',
	X =  -12.715  mm,	Y =   -614.416  mm,	Z =   -242.291  mm,
	W =  90.000 deg,	P =   0.000 deg,	R =   90.000 deg
};
P[2033]{
   GP1:
	UF : 0, UT : 6,		CONFIG : 'N U T, 0, 0, 0',
	X =  -11.258  mm,	Y =   -617.089  mm,	Z =   -242.084  mm,
	W =  90.000 deg,	P =   0.000 deg,	R =   90.000 deg
};
P[2034]{
   GP1:
	UF : 0, UT : 6,		CONFIG : 'N U T, 0, 0, 0',
	X =  -10.750  mm,	Y =   -617.862  mm,	Z =   -242.231  mm,
	W =  90.000 deg,	P =   0.000 deg,	R =   90.000 deg
};
P[2035]{
   GP1:
	UF : 0, UT : 6,		CONFIG : 'N U T, 0, 0, 0',
	X =  -7.433  mm,	Y =   -623.665  mm,	Z =   -242.151  mm,
	W =  90.000 deg,	P =   0.000 deg,	R =   90.000 deg
};
P[2036]{
   GP1:
	UF : 0, UT : 6,		CONFIG : 'N U T, 0, 0, 0',
	X =  -6.987  mm,	Y =   -624.577  mm,	Z =   -241.955  mm,
	W =  90.000 deg,	P =   0.000 deg,	R =   90.000 deg
};
P[2037]{
   GP1:
	UF : 0, UT : 6,		CONFIG : 'N U T, 0, 0, 0',
	X =  -6.074  mm,	Y =   -625.854  mm,	Z =   -242.382  mm,
	W =  90.000 deg,	P =   0.000 deg,	R =   90.000 deg
};
P[2038]{
   GP1:
	UF : 0, UT : 6,		CONFIG : 'N U T, 0, 0, 0',
	X =  -5.550  mm,	Y =   -626.765  mm,	Z =   -242.377  mm,
	W =  90.000 deg,	P =   0.000 deg,	R =   90.000 deg
};
P[2039]{
   GP1:
	UF : 0, UT : 6,		CONFIG : 'N U T, 0, 0, 0',
	X =  -3.732  mm,	Y =   -629.936  mm,	Z =   -242.343  mm,
	W =  90.000 deg,	P =   0.000 deg,	R =   90.000 deg
};
P[2040]{
   GP1:
	UF : 0, UT : 6,		CONFIG : 'N U T, 0, 0, 0',
	X =  -2.993  mm,	Y =   -631.248  mm,	Z =   -242.298  mm,
	W =  90.000 deg,	P =   0.000 deg,	R =   90.000 deg
};
P[2041]{
   GP1:
	UF : 0, UT : 6,		CONFIG : 'N U T, 0, 0, 0',
	X =  0.385  mm,	Y =   -637.197  mm,	Z =   -242.161  mm,
	W =  90.000 deg,	P =   0.000 deg,	R =   90.000 deg
};
P[2042]{
   GP1:
	UF : 0, UT : 6,		CONFIG : 'N U T, 0, 0, 0',
	X =  0.720  mm,	Y =   -637.894  mm,	Z =   -241.997  mm,
	W =  90.000 deg,	P =   0.000 deg,	R =   90.000 deg
};
P[2043]{
   GP1:
	UF : 0, UT : 6,		CONFIG : 'N U T, 0, 0, 0',
	X =  3.294  mm,	Y =   -642.130  mm,	Z =   -242.310  mm,
	W =  90.000 deg,	P =   0.000 deg,	R =   90.000 deg
};
P[2044]{
   GP1:
	UF : 0, UT : 6,		CONFIG : 'N U T, 0, 0, 0',
	X =  3.587  mm,	Y =   -642.922  mm,	Z =   -241.910  mm,
	W =  90.000 deg,	P =   0.000 deg,	R =   90.000 deg
};
P[2045]{
   GP1:
	UF : 0, UT : 6,		CONFIG : 'N U T, 0, 0, 0',
	X =  4.405  mm,	Y =   -644.015  mm,	Z =   -242.364  mm,
	W =  90.000 deg,	P =   0.000 deg,	R =   90.000 deg
};
P[2046]{
   GP1:
	UF : 0, UT : 6,		CONFIG : 'N U T, 0, 0, 0',
	X =  5.198  mm,	Y =   -645.591  mm,	Z =   -242.079  mm,
	W =  90.000 deg,	P =   0.000 deg,	R =   90.000 deg
};
P[2047]{
   GP1:
	UF : 0, UT : 6,		CONFIG : 'N U T, 0, 0, 0',
	X =  6.501  mm,	Y =   -647.766  mm,	Z =   -242.196  mm,
	W =  90.000 deg,	P =   0.000 deg,	R =   90.000 deg
};
P[2048]{
   GP1:
	UF : 0, UT : 6,		CONFIG : 'N U T, 0, 0, 0',
	X =  7.361  mm,	Y =   -649.400  mm,	Z =   -241.992  mm,
	W =  90.000 deg,	P =   0.000 deg,	R =   90.000 deg
};
P[2049]{
   GP1:
	UF : 0, UT : 6,		CONFIG : 'N U T, 0, 0, 0',
	X =  8.202  mm,	Y =   -650.581  mm,	Z =   -242.379  mm,
	W =  90.000 deg,	P =   0.000 deg,	R =   90.000 deg
};
P[2050]{
   GP1:
	UF : 0, UT : 6,		CONFIG : 'N U T, 0, 0, 0',
	X =  8.583  mm,	Y =   -651.558  mm,	Z =   -241.933  mm,
	W =  90.000 deg,	P =   0.000 deg,	R =   90.000 deg
};
P[2051]{
   GP1:
	UF : 0, UT : 6,		CONFIG : 'N U T, 0, 0, 0',
	X =  10.237  mm,	Y =   -654.201  mm,	Z =   -242.245  mm,
	W =  90.000 deg,	P =   0.000 deg,	R =   90.000 deg
};
P[2052]{
   GP1:
	UF : 0, UT : 6,		CONFIG : 'N U T, 0, 0, 0',
	X =  11.788  mm,	Y =   -656.821  mm,	Z =   -242.337  mm,
	W =  90.000 deg,	P =   0.000 deg,	R =   90.000 deg
};
P[2053]{
   GP1:
	UF : 0, UT : 6,		CONFIG : 'N U T, 0, 0, 0',
	X =  12.486  mm,	Y =   -658.185  mm,	Z =   -242.118  mm,
	W =  90.000 deg,	P =   0.000 deg,	R =   90.000 deg
};
P[2054]{
   GP1:
	UF : 0, UT : 6,		CONFIG : 'N U T, 0, 0, 0',
	X =  14.678  mm,	Y =   -661.876  mm,	Z =   -242.266  mm,
	W =  90.000 deg,	P =   0.000 deg,	R =   90.000 deg
};
P[2055]{
   GP1:
	UF : 0, UT : 6,		CONFIG : 'N U T, 0, 0, 0',
	X =  15.897  mm,	Y =   -663.911  mm,	Z =   -242.374  mm,
	W =  90.000 deg,	P =   0.000 deg,	R =   90.000 deg
};
P[2056]{
   GP1:
	UF : 0, UT : 6,		CONFIG : 'N U T, 0, 0, 0',
	X =  16.987  mm,	Y =   -665.910  mm,	Z =   -242.219  mm,
	W =  90.000 deg,	P =   0.000 deg,	R =   90.000 deg
};
P[2057]{
   GP1:
	UF : 0, UT : 6,		CONFIG : 'N U T, 0, 0, 0',
	X =  17.561  mm,	Y =   -666.845  mm,	Z =   -242.299  mm,
	W =  90.000 deg,	P =   0.000 deg,	R =   90.000 deg
};
P[2058]{
   GP1:
	UF : 0, UT : 6,		CONFIG : 'N U T, 0, 0, 0',
	X =  22.129  mm,	Y =   -674.988  mm,	Z =   -241.975  mm,
	W =  90.000 deg,	P =   0.000 deg,	R =   90.000 deg
};
P[2059]{
   GP1:
	UF : 0, UT : 6,		CONFIG : 'N U T, 0, 0, 0',
	X =  23.031  mm,	Y =   -676.453  mm,	Z =   -242.113  mm,
	W =  90.000 deg,	P =   0.000 deg,	R =   90.000 deg
};
P[2060]{
   GP1:
	UF : 0, UT : 6,		CONFIG : 'N U T, 0, 0, 0',
	X =  23.433  mm,	Y =   -677.006  mm,	Z =   -242.313  mm,
	W =  90.000 deg,	P =   0.000 deg,	R =   90.000 deg
};
P[2061]{
   GP1:
	UF : 0, UT : 6,		CONFIG : 'N U T, 0, 0, 0',
	X =  24.005  mm,	Y =   -677.978  mm,	Z =   -242.340  mm,
	W =  90.000 deg,	P =   0.000 deg,	R =   90.000 deg
};
P[2062]{
   GP1:
	UF : 0, UT : 6,		CONFIG : 'N U T, 0, 0, 0',
	X =  24.311  mm,	Y =   -678.617  mm,	Z =   -242.186  mm,
	W =  90.000 deg,	P =   0.000 deg,	R =   90.000 deg
};
P[2063]{
   GP1:
	UF : 0, UT : 6,		CONFIG : 'N U T, 0, 0, 0',
	X =  25.799  mm,	Y =   -681.278  mm,	Z =   -242.069  mm,
	W =  90.000 deg,	P =   0.000 deg,	R =   90.000 deg
};
P[2064]{
   GP1:
	UF : 0, UT : 6,		CONFIG : 'N U T, 0, 0, 0',
	X =  27.323  mm,	Y =   -683.806  mm,	Z =   -242.226  mm,
	W =  90.000 deg,	P =   0.000 deg,	R =   90.000 deg
};
P[2065]{
   GP1:
	UF : 0, UT : 6,		CONFIG : 'N U T, 0, 0, 0',
	X =  28.261  mm,	Y =   -685.424  mm,	Z =   -242.235  mm,
	W =  90.000 deg,	P =   0.000 deg,	R =   90.000 deg
};
P[2066]{
   GP1:
	UF : 0, UT : 6,		CONFIG : 'N U T, 0, 0, 0',
	X =  31.573  mm,	Y =   -691.087  mm,	Z =   -242.338  mm,
	W =  90.000 deg,	P =   0.000 deg,	R =   90.000 deg
};
P[2067]{
   GP1:
	UF : 0, UT : 6,		CONFIG : 'N U T, 0, 0, 0',
	X =  33.251  mm,	Y =   -694.098  mm,	Z =   -242.189  mm,
	W =  90.000 deg,	P =   0.000 deg,	R =   90.000 deg
};
P[2068]{
   GP1:
	UF : 0, UT : 6,		CONFIG : 'N U T, 0, 0, 0',
	X =  35.434  mm,	Y =   -697.894  mm,	Z =   -242.167  mm,
	W =  90.000 deg,	P =   0.000 deg,	R =   90.000 deg
};
P[2069]{
   GP1:
	UF : 0, UT : 6,		CONFIG : 'N U T, 0, 0, 0',
	X =  36.268  mm,	Y =   -699.147  mm,	Z =   -242.277  mm,
	W =  90.000 deg,	P =   0.000 deg,	R =   90.000 deg
};
P[2070]{
   GP1:
	UF : 0, UT : 6,		CONFIG : 'N U T, 0, 0, 0',
	X =  36.615  mm,	Y =   -699.653  mm,	Z =   -242.253  mm,
	W =  90.000 deg,	P =   0.000 deg,	R =   90.000 deg
};
P[2071]{
   GP1:
	UF : 0, UT : 6,		CONFIG : 'N U T, 0, 0, 0',
	X =  37.878  mm,	Y =   -701.299  mm,	Z =   -242.243  mm,
	W =  90.000 deg,	P =   0.000 deg,	R =   90.000 deg
};
P[2072]{
   GP1:
	UF : 0, UT : 6,		CONFIG : 'N U T, 0, 0, 0',
	X =  39.141  mm,	Y =   -702.440  mm,	Z =   -242.302  mm,
	W =  90.000 deg,	P =   0.000 deg,	R =   90.000 deg
};
P[2073]{
   GP1:
	UF : 0, UT : 6,		CONFIG : 'N U T, 0, 0, 0',
	X =  39.757  mm,	Y =   -703.129  mm,	Z =   -242.058  mm,
	W =  90.000 deg,	P =   0.000 deg,	R =   90.000 deg
};
P[2074]{
   GP1:
	UF : 0, UT : 6,		CONFIG : 'N U T, 0, 0, 0',
	X =  40.555  mm,	Y =   -703.641  mm,	Z =   -242.050  mm,
	W =  90.000 deg,	P =   0.000 deg,	R =   90.000 deg
};
P[2075]{
   GP1:
	UF : 0, UT : 6,		CONFIG : 'N U T, 0, 0, 0',
	X =  42.095  mm,	Y =   -704.383  mm,	Z =   -242.283  mm,
	W =  90.000 deg,	P =   0.000 deg,	R =   90.000 deg
};
P[2076]{
   GP1:
	UF : 0, UT : 6,		CONFIG : 'N U T, 0, 0, 0',
	X =  43.715  mm,	Y =   -705.086  mm,	Z =   -242.143  mm,
	W =  90.000 deg,	P =   0.000 deg,	R =   90.000 deg
};
P[2077]{
   GP1:
	UF : 0, UT : 6,		CONFIG : 'N U T, 0, 0, 0',
	X =  44.374  mm,	Y =   -705.169  mm,	Z =   -242.322  mm,
	W =  90.000 deg,	P =   0.000 deg,	R =   90.000 deg
};
P[2078]{
   GP1:
	UF : 0, UT : 6,		CONFIG : 'N U T, 0, 0, 0',
	X =  47.959  mm,	Y =   -705.580  mm,	Z =   -242.346  mm,
	W =  90.000 deg,	P =   0.000 deg,	R =   90.000 deg
};
P[2079]{
   GP1:
	UF : 0, UT : 6,		CONFIG : 'N U T, 0, 0, 0',
	X =  54.236  mm,	Y =   -704.008  mm,	Z =   -242.165  mm,
	W =  90.000 deg,	P =   0.000 deg,	R =   90.000 deg
};
P[2080]{
   GP1:
	UF : 0, UT : 6,		CONFIG : 'N U T, 0, 0, 0',
	X =  56.953  mm,	Y =   -702.428  mm,	Z =   -242.346  mm,
	W =  90.000 deg,	P =   0.000 deg,	R =   90.000 deg
};
P[2081]{
   GP1:
	UF : 0, UT : 6,		CONFIG : 'N U T, 0, 0, 0',
	X =  60.997  mm,	Y =   -700.098  mm,	Z =   -242.336  mm,
	W =  90.000 deg,	P =   0.000 deg,	R =   90.000 deg
};
P[2082]{
   GP1:
	UF : 0, UT : 6,		CONFIG : 'N U T, 0, 0, 0',
	X =  61.889  mm,	Y =   -699.572  mm,	Z =   -242.362  mm,
	W =  90.000 deg,	P =   0.000 deg,	R =   90.000 deg
};
P[2083]{
   GP1:
	UF : 0, UT : 6,		CONFIG : 'N U T, 0, 0, 0',
	X =  63.628  mm,	Y =   -698.590  mm,	Z =   -242.310  mm,
	W =  90.000 deg,	P =   0.000 deg,	R =   90.000 deg
};
P[2084]{
   GP1:
	UF : 0, UT : 6,		CONFIG : 'N U T, 0, 0, 0',
	X =  65.682  mm,	Y =   -697.518  mm,	Z =   -242.033  mm,
	W =  90.000 deg,	P =   0.000 deg,	R =   90.000 deg
};
P[2085]{
   GP1:
	UF : 0, UT : 6,		CONFIG : 'N U T, 0, 0, 0',
	X =  72.768  mm,	Y =   -693.486  mm,	Z =   -241.890  mm,
	W =  90.000 deg,	P =   0.000 deg,	R =   90.000 deg
};
P[2086]{
   GP1:
	UF : 0, UT : 6,		CONFIG : 'N U T, 0, 0, 0',
	X =  73.444  mm,	Y =   -692.992  mm,	Z =   -242.140  mm,
	W =  90.000 deg,	P =   0.000 deg,	R =   90.000 deg
};
P[2087]{
   GP1:
	UF : 0, UT : 6,		CONFIG : 'N U T, 0, 0, 0',
	X =  74.560  mm,	Y =   -692.300  mm,	Z =   -242.256  mm,
	W =  90.000 deg,	P =   0.000 deg,	R =   90.000 deg
};
P[2088]{
   GP1:
	UF : 0, UT : 6,		CONFIG : 'N U T, 0, 0, 0',
	X =  75.813  mm,	Y =   -691.656  mm,	Z =   -242.064  mm,
	W =  90.000 deg,	P =   0.000 deg,	R =   90.000 deg
};
P[2089]{
   GP1:
	UF : 0, UT : 6,		CONFIG : 'N U T, 0, 0, 0',
	X =  77.316  mm,	Y =   -690.716  mm,	Z =   -242.239  mm,
	W =  90.000 deg,	P =   0.000 deg,	R =   90.000 deg
};
P[2090]{
   GP1:
	UF : 0, UT : 6,		CONFIG : 'N U T, 0, 0, 0',
	X =  78.337  mm,	Y =   -690.185  mm,	Z =   -242.097  mm,
	W =  90.000 deg,	P =   0.000 deg,	R =   90.000 deg
};
P[2091]{
   GP1:
	UF : 0, UT : 6,		CONFIG : 'N U T, 0, 0, 0',
	X =  81.339  mm,	Y =   -688.441  mm,	Z =   -242.122  mm,
	W =  90.000 deg,	P =   0.000 deg,	R =   90.000 deg
};
P[2092]{
   GP1:
	UF : 0, UT : 6,		CONFIG : 'N U T, 0, 0, 0',
	X =  82.336  mm,	Y =   -687.870  mm,	Z =   -242.110  mm,
	W =  90.000 deg,	P =   0.000 deg,	R =   90.000 deg
};
P[2093]{
   GP1:
	UF : 0, UT : 6,		CONFIG : 'N U T, 0, 0, 0',
	X =  82.896  mm,	Y =   -687.463  mm,	Z =   -242.311  mm,
	W =  90.000 deg,	P =   0.000 deg,	R =   90.000 deg
};
P[2094]{
   GP1:
	UF : 0, UT : 6,		CONFIG : 'N U T, 0, 0, 0',
	X =  86.660  mm,	Y =   -685.342  mm,	Z =   -242.185  mm,
	W =  90.000 deg,	P =   0.000 deg,	R =   90.000 deg
};
P[2095]{
   GP1:
	UF : 0, UT : 6,		CONFIG : 'N U T, 0, 0, 0',
	X =  91.888  mm,	Y =   -682.256  mm,	Z =   -242.349  mm,
	W =  90.000 deg,	P =   0.000 deg,	R =   90.000 deg
};
P[2096]{
   GP1:
	UF : 0, UT : 6,		CONFIG : 'N U T, 0, 0, 0',
	X =  96.389  mm,	Y =   -679.778  mm,	Z =   -242.059  mm,
